LIN {X 0,Y 269.134,Z 589.137,A -85,B 0,C 180,E1 -17739.772,E2 -17739.772} C_VEL
LIN {X 0,Y 269.562,Z 582.717,A -85,B 0,C 180,E1 -17742.421,E2 -17742.421} C_VEL
LIN {X 0,Y 270.303,Z 575.756,A -85,B 0,C 180,E1 -17744.685,E2 -17744.685} C_VEL
LIN {X 0,Y 271.369,Z 568.724,A -85,B 0,C 180,E1 -17746.551,E2 -17746.551} C_VEL
LIN {X 0,Y 272.807,Z 560.299,A -85,B 0,C 180,E1 -17748.396,E2 -17748.396} C_VEL
LIN {X 0,Y 273.728,Z 553.275,A -85,B 0,C 180,E1 -17749.693,E2 -17749.693} C_VEL
LIN {X 0,Y 274.219,Z 542.305,A -85,B 0,C 180,E1 -17751.421,E2 -17751.421} C_VEL
LIN {X 0,Y 274.396,Z 531.867,A -85,B 0,C 180,E1 -17752.772,E2 -17752.772} C_VEL
LIN {X 0,Y 274.061,Z 519.052,A -85,B 0,C 180,E1 -17754.123,E2 -17754.123} C_VEL
LIN {X 0,Y 272.996,Z 505.88,A -85,B 0,C 180,E1 -17755.219,E2 -17755.219} C_VEL
LIN {X 0,Y 270.997,Z 492.141,A -85,B 0,C 180,E1 -17756.117,E2 -17756.117} C_VEL
LIN {X 0,Y 270.32,Z 487.569,A -85,B 0,C 180,E1 -17756.386,E2 -17756.386} C_VEL
LIN {X 0,Y 271.834,Z 476.288,A -85,B 0,C 180,E1 -17761.441,E2 -17761.441} C_VEL
LIN {X 0,Y 273.235,Z 467.638,A -85,B 0,C 180,E1 -17765.36,E2 -17765.36} C_VEL
LIN {X 0,Y 274.283,Z 461.982,A -85,B 0,C 180,E1 -17767.948,E2 -17767.948} C_VEL
LIN {X 0,Y 274.444,Z 460.134,A -85,B 0,C 180,E1 -17768.812,E2 -17768.812} C_VEL
LIN {X 0,Y 273.389,Z 453.927,A -85,B 0,C 180,E1 -17771.942,E2 -17771.942} C_VEL
LIN {X 0,Y 272.317,Z 448.311,A -85,B 0,C 180,E1 -17774.934,E2 -17774.934} C_VEL
LIN {X 0,Y 270.924,Z 441.471,A -85,B 0,C 180,E1 -17778.788,E2 -17778.788} C_VEL
LIN {X 0,Y 270.195,Z 437.829,A -85,B 0,C 180,E1 -17781.026,E2 -17781.026} C_VEL
LIN {X 0,Y 270.255,Z 437.821,A -85,B 0,C 180,E1 -17783.722,E2 -17783.722} C_VEL
LIN {X 0,Y 270.204,Z 437.829,A -85,B 0,C 180,E1 -17786.893,E2 -17786.893} C_VEL
LIN {X 0,Y 270.195,Z 437.83,A -85,B 0,C 180,E1 -17790.383,E2 -17790.383} C_VEL
LIN {X 0,Y 270.262,Z 437.819,A -85,B 0,C 180,E1 -17793.764,E2 -17793.764} C_VEL
LIN {X 0,Y 270.237,Z 437.822,A -85,B 0,C 180,E1 -17797.039,E2 -17797.039} C_VEL
LIN {X 0,Y 270.303,Z 437.818,A -85,B 0,C 180,E1 -17800.245,E2 -17800.245} C_VEL
LIN {X 0,Y 270.404,Z 437.802,A -85,B 0,C 180,E1 -17804.936,E2 -17804.936} C_VEL
LIN {X 0,Y 270.413,Z 437.801,A -85,B 0,C 180,E1 -17809.518,E2 -17809.518} C_VEL
LIN {X 0,Y 270.586,Z 437.779,A -85,B 0,C 180,E1 -17812.538,E2 -17812.538} C_VEL
LIN {X 0,Y 270.789,Z 437.753,A -85,B 0,C 180,E1 -17818.513,E2 -17818.513} C_VEL
LIN {X 0,Y 270.788,Z 437.752,A -85,B 0,C 180,E1 -17821.487,E2 -17821.487} C_VEL
LIN {X 0,Y 270.613,Z 437.771,A -85,B 0,C 180,E1 -17827.461,E2 -17827.461} C_VEL
LIN {X 0,Y 270.443,Z 437.795,A -85,B 0,C 180,E1 -17830.481,E2 -17830.481} C_VEL
LIN {X 0,Y 270.404,Z 437.798,A -85,B 0,C 180,E1 -17835.065,E2 -17835.065} C_VEL
LIN {X 0,Y 270.303,Z 437.806,A -85,B 0,C 180,E1 -17839.756,E2 -17839.756} C_VEL
LIN {X 0,Y 270.275,Z 437.81,A -85,B 0,C 180,E1 -17844.586,E2 -17844.586} C_VEL
LIN {X 0,Y 270.271,Z 437.821,A -85,B 0,C 180,E1 -17847.909,E2 -17847.909} C_VEL
LIN {X 0,Y 270.185,Z 437.823,A -85,B 0,C 180,E1 -17851.349,E2 -17851.349} C_VEL
LIN {X 0,Y 270.216,Z 437.817,A -85,B 0,C 180,E1 -17854.904,E2 -17854.904} C_VEL
LIN {X 0,Y 270.223,Z 437.822,A -85,B 0,C 180,E1 -17858.717,E2 -17858.717} C_VEL
LIN {X 0,Y 270.166,Z 437.829,A -85,B 0,C 180,E1 -17863.249,E2 -17863.249} C_VEL
LIN {X 0,Y 270.173,Z 437.829,A -85,B 0,C 180,E1 -17867.442,E2 -17867.442} C_VEL
LIN {X 0,Y 270.209,Z 437.823,A -85,B 0,C 180,E1 -17871.375,E2 -17871.375} C_VEL
LIN {X 0,Y 270.217,Z 437.819,A -85,B 0,C 180,E1 -17875.097,E2 -17875.097} C_VEL
LIN {X 0,Y 270.203,Z 437.825,A -85,B 0,C 180,E1 -17879.131,E2 -17879.131} C_VEL
LIN {X 0,Y 270.273,Z 437.816,A -85,B 0,C 180,E1 -17882.144,E2 -17882.144} C_VEL
LIN {X 0,Y 270.28,Z 437.813,A -85,B 0,C 180,E1 -17885.519,E2 -17885.519} C_VEL
LIN {X 0,Y 270.267,Z 437.861,A -85,B 0,C 180,E1 -17887.826,E2 -17887.826} C_VEL
LIN {X 0,Y 274.013,Z 447.701,A -85,B 0,C 180,E1 -17889.063,E2 -17889.063} C_VEL
LIN {X 0,Y 277.349,Z 457.508,A -85,B 0,C 180,E1 -17890.474,E2 -17890.474} C_VEL
LIN {X 0,Y 279.974,Z 467.572,A -85,B 0,C 180,E1 -17892.105,E2 -17892.105} C_VEL
LIN {X 0,Y 278.962,Z 475.715,A -85,B 0,C 180,E1 -17893.348,E2 -17893.348} C_VEL
LIN {X 0,Y 277.223,Z 486.274,A -85,B 0,C 180,E1 -17895.315,E2 -17895.315} C_VEL
LIN {X 0,Y 275.79,Z 494.07,A -85,B 0,C 180,E1 -17897.116,E2 -17897.116} C_VEL
LIN {X 0,Y 274.344,Z 501.7,A -85,B 0,C 180,E1 -17899.297,E2 -17899.297} C_VEL
LIN {X 0,Y 273.311,Z 506.88,A -85,B 0,C 180,E1 -17901.125,E2 -17901.125} C_VEL
LIN {X 0,Y 272.448,Z 511.909,A -85,B 0,C 180,E1 -17903.334,E2 -17903.334} C_VEL
LIN {X 0,Y 271.535,Z 515.856,A -85,B 0,C 180,E1 -17905.547,E2 -17905.547} C_VEL
LIN {X 0,Y 271.094,Z 517.898,A -85,B 0,C 180,E1 -17907.028,E2 -17907.028} C_VEL
LIN {X 0,Y 270.698,Z 520.727,A -85,B 0,C 180,E1 -17910,E2 -17910} C_VEL
LIN {X 0,Y 270.688,Z 521.555,A -85,B 0,C 180,E1 -17911.488,E2 -17911.488} C_VEL
LIN {X 0,Y 270.509,Z 522.06,A -85,B 0,C 180,E1 -17914.471,E2 -17914.471} C_VEL
LIN {X 0,Y 271.194,Z 521.003,A -85,B 0,C 180,E1 -17917.445,E2 -17917.445} C_VEL
LIN {X 0,Y 271.754,Z 519.845,A -85,B 0,C 180,E1 -17918.927,E2 -17918.927} C_VEL
LIN {X 0,Y 272.834,Z 516.501,A -85,B 0,C 180,E1 -17921.802,E2 -17921.802} C_VEL
LIN {X 0,Y 273.931,Z 512.606,A -85,B 0,C 180,E1 -17924.107,E2 -17924.107} C_VEL
LIN {X 0,Y 275.118,Z 507.732,A -85,B 0,C 180,E1 -17926.32,E2 -17926.32} C_VEL
LIN {X 0,Y 276.586,Z 501.563,A -85,B 0,C 180,E1 -17928.52,E2 -17928.52} C_VEL
LIN {X 0,Y 278.443,Z 493.783,A -85,B 0,C 180,E1 -17930.694,E2 -17930.694} C_VEL
LIN {X 0,Y 280.202,Z 485.823,A -85,B 0,C 180,E1 -17932.489,E2 -17932.489} C_VEL
LIN {X 0,Y 281.896,Z 476.106,A -85,B 0,C 180,E1 -17934.291,E2 -17934.291} C_VEL
LIN {X 0,Y 282.425,Z 472.703,A -85,B 0,C 180,E1 -17934.83,E2 -17934.83} C_VEL
LIN {X 0,Y 279.934,Z 463.035,A -85,B 0,C 180,E1 -17936.62,E2 -17936.62} C_VEL
LIN {X 0,Y 276.46,Z 452.721,A -85,B 0,C 180,E1 -17938.332,E2 -17938.332} C_VEL
LIN {X 0,Y 272.01,Z 442.14,A -85,B 0,C 180,E1 -17939.923,E2 -17939.923} C_VEL
LIN {X 0,Y 270.458,Z 438.953,A -85,B 0,C 180,E1 -17940.387,E2 -17940.387} C_VEL
LIN {X 0,Y 270.228,Z 437.825,A -85,B 0,C 180,E1 -17940.537,E2 -17940.537} C_VEL
LIN {X 0,Y 270.219,Z 437.824,A -85,B 0,C 180,E1 -17944.904,E2 -17944.904} C_VEL
LIN {X 0,Y 270.226,Z 437.824,A -85,B 0,C 180,E1 -17948.717,E2 -17948.717} C_VEL
LIN {X 0,Y 270.169,Z 437.83,A -85,B 0,C 180,E1 -17953.249,E2 -17953.249} C_VEL
LIN {X 0,Y 270.175,Z 437.827,A -85,B 0,C 180,E1 -17957.442,E2 -17957.442} C_VEL
LIN {X 0,Y 270.21,Z 437.823,A -85,B 0,C 180,E1 -17961.374,E2 -17961.374} C_VEL
LIN {X 0,Y 270.218,Z 437.822,A -85,B 0,C 180,E1 -17965.097,E2 -17965.097} C_VEL
LIN {X 0,Y 270.204,Z 437.825,A -85,B 0,C 180,E1 -17969.13,E2 -17969.13} C_VEL
LIN {X 0,Y 270.269,Z 437.818,A -85,B 0,C 180,E1 -17972.145,E2 -17972.145} C_VEL
LIN {X 0,Y 270.242,Z 437.821,A -85,B 0,C 180,E1 -17975.537,E2 -17975.537} C_VEL
LIN {X 0,Y 270.36,Z 437.805,A -85,B 0,C 180,E1 -17980.841,E2 -17980.841} C_VEL
LIN {X 0,Y 270.415,Z 437.929,A -85,B 0,C 180,E1 -17980.993,E2 -17980.993} C_VEL
LIN {X 0,Y 273.457,Z 451.257,A -85,B 0,C 180,E1 -17982.473,E2 -17982.473} C_VEL
LIN {X 0,Y 274.58,Z 456.844,A -85,B 0,C 180,E1 -17983.195,E2 -17983.195} C_VEL
LIN {X 0,Y 273.669,Z 469.268,A -85,B 0,C 180,E1 -17984.929,E2 -17984.929} C_VEL
LIN {X 0,Y 272.809,Z 479.061,A -85,B 0,C 180,E1 -17986.593,E2 -17986.593} C_VEL
LIN {X 0,Y 271.9,Z 490.128,A -85,B 0,C 180,E1 -17988.897,E2 -17988.897} C_VEL
LIN {X 0,Y 271.19,Z 498.55,A -85,B 0,C 180,E1 -17991.054,E2 -17991.054} C_VEL
LIN {X 0,Y 270.61,Z 506.844,A -85,B 0,C 180,E1 -17993.663,E2 -17993.663} C_VEL
LIN {X 0,Y 270.176,Z 513.358,A -85,B 0,C 180,E1 -17996.271,E2 -17996.271} C_VEL
LIN {X 0,Y 270.262,Z 517.749,A -85,B 0,C 180,E1 -17998.51,E2 -17998.51} C_VEL
LIN {X 0,Y 270.571,Z 520.097,A -85,B 0,C 180,E1 -18000,E2 -18000} C_VEL
LIN {X 0,Y 270.747,Z 522.029,A -85,B 0,C 180,E1 -18001.487,E2 -18001.487} C_VEL
LIN {X 0,Y 271.393,Z 524.678,A -85,B 0,C 180,E1 -18004.455,E2 -18004.455} C_VEL
LIN {X 0,Y 271.923,Z 525.431,A -85,B 0,C 180,E1 -18005.934,E2 -18005.934} C_VEL
LIN {X 0,Y 273.501,Z 525.662,A -85,B 0,C 180,E1 -18008.869,E2 -18008.869} C_VEL
LIN {X 0,Y 275.601,Z 524.401,A -85,B 0,C 180,E1 -18011.771,E2 -18011.771} C_VEL
LIN {X 0,Y 276.765,Z 523.168,A -85,B 0,C 180,E1 -18013.211,E2 -18013.211} C_VEL
LIN {X 0,Y 279.498,Z 519.777,A -85,B 0,C 180,E1 -18015.867,E2 -18015.867} C_VEL
LIN {X 0,Y 280.197,Z 518.177,A -85,B 0,C 180,E1 -18017.024,E2 -18017.024} C_VEL
LIN {X 0,Y 279.908,Z 515.583,A -85,B 0,C 180,E1 -18018.982,E2 -18018.982} C_VEL
LIN {X 0,Y 279.846,Z 512.387,A -85,B 0,C 180,E1 -18020.895,E2 -18020.895} C_VEL
LIN {X 0,Y 280.862,Z 509.845,A -85,B 0,C 180,E1 -18021.959,E2 -18021.959} C_VEL
LIN {X 0,Y 285.102,Z 501.844,A -85,B 0,C 180,E1 -18024.387,E2 -18024.387} C_VEL
LIN {X 0,Y 288.996,Z 493.552,A -85,B 0,C 180,E1 -18026.348,E2 -18026.348} C_VEL
LIN {X 0,Y 289.688,Z 491.994,A -85,B 0,C 180,E1 -18026.668,E2 -18026.668} C_VEL
LIN {X 0,Y 289.831,Z 489.623,A -85,B 0,C 180,E1 -18027.434,E2 -18027.434} C_VEL
LIN {X 0,Y 289.235,Z 483.398,A -85,B 0,C 180,E1 -18029.77,E2 -18029.77} C_VEL
LIN {X 0,Y 288.163,Z 478.273,A -85,B 0,C 180,E1 -18031.983,E2 -18031.983} C_VEL
LIN {X 0,Y 286.822,Z 473.819,A -85,B 0,C 180,E1 -18034.303,E2 -18034.303} C_VEL
LIN {X 0,Y 285.403,Z 471.506,A -85,B 0,C 180,E1 -18036.228,E2 -18036.228} C_VEL
LIN {X 0,Y 284.095,Z 470.015,A -85,B 0,C 180,E1 -18038.203,E2 -18038.203} C_VEL
LIN {X 0,Y 282.968,Z 469.651,A -85,B 0,C 180,E1 -18040.222,E2 -18040.222} C_VEL
LIN {X 0,Y 281.985,Z 470.615,A -85,B 0,C 180,E1 -18042.293,E2 -18042.293} C_VEL
LIN {X 0,Y 281.387,Z 472.597,A -85,B 0,C 180,E1 -18044.374,E2 -18044.374} C_VEL
LIN {X 0,Y 281.101,Z 475.772,A -85,B 0,C 180,E1 -18046.473,E2 -18046.473} C_VEL
LIN {X 0,Y 281.308,Z 479.869,A -85,B 0,C 180,E1 -18048.547,E2 -18048.547} C_VEL
LIN {X 0,Y 281.488,Z 484.367,A -85,B 0,C 180,E1 -18050.198,E2 -18050.198} C_VEL
LIN {X 0,Y 281.102,Z 490.544,A -85,B 0,C 180,E1 -18051.779,E2 -18051.779} C_VEL
LIN {X 0,Y 281.145,Z 493.947,A -85,B 0,C 180,E1 -18052.692,E2 -18052.692} C_VEL
LIN {X 0,Y 280.667,Z 508.223,A -85,B 0,C 180,E1 -18055.919,E2 -18055.919} C_VEL
LIN {X 0,Y 279.754,Z 521.489,A -85,B 0,C 180,E1 -18058.666,E2 -18058.666} C_VEL
LIN {X 0,Y 278.399,Z 532.665,A -85,B 0,C 180,E1 -18060.925,E2 -18060.925} C_VEL
LIN {X 0,Y 276.661,Z 541.8,A -85,B 0,C 180,E1 -18062.79,E2 -18062.79} C_VEL
LIN {X 0,Y 273.354,Z 553.407,A -85,B 0,C 180,E1 -18065.304,E2 -18065.304} C_VEL
LIN {X 0,Y 269.883,Z 564.585,A -85,B 0,C 180,E1 -18068.217,E2 -18068.217} C_VEL
LIN {X 0,Y 266.722,Z 572.712,A -85,B 0,C 180,E1 -18070.769,E2 -18070.769} C_VEL
LIN {X 0,Y 264.622,Z 578.556,A -85,B 0,C 180,E1 -18073.013,E2 -18073.013} C_VEL
LIN {X 0,Y 262.894,Z 584.824,A -85,B 0,C 180,E1 -18076.078,E2 -18076.078} C_VEL
LIN {X 0,Y 262.029,Z 594.375,A -85,B 0,C 180,E1 -18082.293,E2 -18082.293} C_VEL
LIN {X 0,Y 262.433,Z 597.47,A -85,B 0,C 180,E1 -18085.392,E2 -18085.392} C_VEL
LIN {X 0,Y 263.066,Z 598.826,A -85,B 0,C 180,E1 -18088.469,E2 -18088.469} C_VEL
LIN {X 0,Y 263.49,Z 598.901,A -85,B 0,C 180,E1 -18090,E2 -18090} C_VEL
LIN {X 0,Y 263.075,Z 598.446,A -85,B 0,C 180,E1 -18091.53,E2 -18091.53} C_VEL
LIN {X 0,Y 262.734,Z 597.546,A -85,B 0,C 180,E1 -18093.066,E2 -18093.066} C_VEL
LIN {X 0,Y 262.536,Z 596.227,A -85,B 0,C 180,E1 -18094.606,E2 -18094.606} C_VEL
LIN {X 0,Y 262.182,Z 592.821,A -85,B 0,C 180,E1 -18097.335,E2 -18097.335} C_VEL
LIN {X 0,Y 262.066,Z 588.033,A -85,B 0,C 180,E1 -18100.038,E2 -18100.038} C_VEL
LIN {X 0,Y 262.569,Z 581.59,A -85,B 0,C 180,E1 -18102.757,E2 -18102.757} C_VEL
LIN {X 0,Y 263.347,Z 574.603,A -85,B 0,C 180,E1 -18105.082,E2 -18105.082} C_VEL
LIN {X 0,Y 264.607,Z 567.41,A -85,B 0,C 180,E1 -18107.027,E2 -18107.027} C_VEL
LIN {X 0,Y 266.024,Z 559.1,A -85,B 0,C 180,E1 -18108.882,E2 -18108.882} C_VEL
LIN {X 0,Y 266.735,Z 553.115,A -85,B 0,C 180,E1 -18110.031,E2 -18110.031} C_VEL
LIN {X 0,Y 267.308,Z 542.427,A -85,B 0,C 180,E1 -18111.785,E2 -18111.785} C_VEL
LIN {X 0,Y 267.521,Z 530.306,A -85,B 0,C 180,E1 -18113.412,E2 -18113.412} C_VEL
LIN {X 0,Y 267.214,Z 517.51,A -85,B 0,C 180,E1 -18114.782,E2 -18114.782} C_VEL
LIN {X 0,Y 266.029,Z 503.862,A -85,B 0,C 180,E1 -18115.946,E2 -18115.946} C_VEL
LIN {X 0,Y 264.013,Z 490.435,A -85,B 0,C 180,E1 -18116.843,E2 -18116.843} C_VEL
LIN {X 0,Y 263.384,Z 486.54,A -85,B 0,C 180,E1 -18117.083,E2 -18117.083} C_VEL
LIN {X 0,Y 264.969,Z 475.794,A -85,B 0,C 180,E1 -18122.037,E2 -18122.037} C_VEL
LIN {X 0,Y 266.215,Z 468.377,A -85,B 0,C 180,E1 -18125.506,E2 -18125.506} C_VEL
LIN {X 0,Y 267.341,Z 462.21,A -85,B 0,C 180,E1 -18128.423,E2 -18128.423} C_VEL
LIN {X 0,Y 267.076,Z 458.563,A -85,B 0,C 180,E1 -18130.26,E2 -18130.26} C_VEL
LIN {X 0,Y 265.602,Z 450.824,A -85,B 0,C 180,E1 -18134.403,E2 -18134.403} C_VEL
LIN {X 0,Y 264.198,Z 444.015,A -85,B 0,C 180,E1 -18138.315,E2 -18138.315} C_VEL
LIN {X 0,Y 263.159,Z 438.707,A -85,B 0,C 180,E1 -18141.647,E2 -18141.647} C_VEL
LIN {X 0,Y 263.188,Z 438.702,A -85,B 0,C 180,E1 -18144.022,E2 -18144.022} C_VEL
LIN {X 0,Y 263.133,Z 438.71,A -85,B 0,C 180,E1 -18147.712,E2 -18147.712} C_VEL
LIN {X 0,Y 263.196,Z 438.702,A -85,B 0,C 180,E1 -18151.785,E2 -18151.785} C_VEL
LIN {X 0,Y 263.226,Z 438.695,A -85,B 0,C 180,E1 -18155.2,E2 -18155.2} C_VEL
LIN {X 0,Y 263.269,Z 438.693,A -85,B 0,C 180,E1 -18159.694,E2 -18159.694} C_VEL
LIN {X 0,Y 263.352,Z 438.682,A -85,B 0,C 180,E1 -18164.522,E2 -18164.522} C_VEL
LIN {X 0,Y 263.356,Z 438.68,A -85,B 0,C 180,E1 -18169.234,E2 -18169.234} C_VEL
LIN {X 0,Y 263.546,Z 438.658,A -85,B 0,C 180,E1 -18172.338,E2 -18172.338} C_VEL
LIN {X 0,Y 263.753,Z 438.63,A -85,B 0,C 180,E1 -18178.473,E2 -18178.473} C_VEL
LIN {X 0,Y 263.753,Z 438.629,A -85,B 0,C 180,E1 -18181.527,E2 -18181.527} C_VEL
LIN {X 0,Y 263.574,Z 438.649,A -85,B 0,C 180,E1 -18187.662,E2 -18187.662} C_VEL
LIN {X 0,Y 263.375,Z 438.674,A -85,B 0,C 180,E1 -18190.766,E2 -18190.766} C_VEL
LIN {X 0,Y 263.352,Z 438.678,A -85,B 0,C 180,E1 -18195.478,E2 -18195.478} C_VEL
LIN {X 0,Y 263.265,Z 438.677,A -85,B 0,C 180,E1 -18200.307,E2 -18200.307} C_VEL
LIN {X 0,Y 263.209,Z 438.69,A -85,B 0,C 180,E1 -18205.292,E2 -18205.292} C_VEL
LIN {X 0,Y 263.176,Z 438.7,A -85,B 0,C 180,E1 -18208.73,E2 -18208.73} C_VEL
LIN {X 0,Y 263.134,Z 438.691,A -85,B 0,C 180,E1 -18212.289,E2 -18212.289} C_VEL
LIN {X 0,Y 263.189,Z 438.698,A -85,B 0,C 180,E1 -18215.978,E2 -18215.978} C_VEL
LIN {X 0,Y 263.116,Z 438.708,A -85,B 0,C 180,E1 -18219.871,E2 -18219.871} C_VEL
LIN {X 0,Y 263.124,Z 438.705,A -85,B 0,C 180,E1 -18223.985,E2 -18223.985} C_VEL
LIN {X 0,Y 263.126,Z 438.703,A -85,B 0,C 180,E1 -18228.407,E2 -18228.407} C_VEL
LIN {X 0,Y 263.167,Z 438.7,A -85,B 0,C 180,E1 -18232.105,E2 -18232.105} C_VEL
LIN {X 0,Y 263.186,Z 438.701,A -85,B 0,C 180,E1 -18235.891,E2 -18235.891} C_VEL
LIN {X 0,Y 263.156,Z 438.705,A -85,B 0,C 180,E1 -18239.508,E2 -18239.508} C_VEL
LIN {X 0,Y 263.2,Z 438.699,A -85,B 0,C 180,E1 -18243.004,E2 -18243.004} C_VEL
LIN {X 0,Y 263.201,Z 438.7,A -85,B 0,C 180,E1 -18247.118,E2 -18247.118} C_VEL
LIN {X 0,Y 265.506,Z 444.774,A -85,B 0,C 180,E1 -18247.891,E2 -18247.891} C_VEL
LIN {X 0,Y 269.502,Z 455.525,A -85,B 0,C 180,E1 -18249.44,E2 -18249.44} C_VEL
LIN {X 0,Y 272.313,Z 465.51,A -85,B 0,C 180,E1 -18251.042,E2 -18251.042} C_VEL
LIN {X 0,Y 273.33,Z 470.093,A -85,B 0,C 180,E1 -18251.846,E2 -18251.846} C_VEL
LIN {X 0,Y 271.785,Z 480.105,A -85,B 0,C 180,E1 -18253.475,E2 -18253.475} C_VEL
LIN {X 0,Y 270.111,Z 489.175,A -85,B 0,C 180,E1 -18255.305,E2 -18255.305} C_VEL
LIN {X 0,Y 268.419,Z 497.955,A -85,B 0,C 180,E1 -18257.526,E2 -18257.526} C_VEL
LIN {X 0,Y 266.995,Z 505.021,A -85,B 0,C 180,E1 -18259.766,E2 -18259.766} C_VEL
LIN {X 0,Y 266.136,Z 509.77,A -85,B 0,C 180,E1 -18261.649,E2 -18261.649} C_VEL
LIN {X 0,Y 265.108,Z 514.417,A -85,B 0,C 180,E1 -18263.913,E2 -18263.913} C_VEL
LIN {X 0,Y 264.312,Z 517.986,A -85,B 0,C 180,E1 -18266.189,E2 -18266.189} C_VEL
LIN {X 0,Y 263.798,Z 520.564,A -85,B 0,C 180,E1 -18268.474,E2 -18268.474} C_VEL
LIN {X 0,Y 263.663,Z 522.584,A -85,B 0,C 180,E1 -18271.528,E2 -18271.528} C_VEL
LIN {X 0,Y 263.495,Z 523.068,A -85,B 0,C 180,E1 -18274.59,E2 -18274.59} C_VEL
LIN {X 0,Y 264.223,Z 521.986,A -85,B 0,C 180,E1 -18277.643,E2 -18277.643} C_VEL
LIN {X 0,Y 264.811,Z 520.814,A -85,B 0,C 180,E1 -18279.163,E2 -18279.163} C_VEL
LIN {X 0,Y 265.909,Z 517.522,A -85,B 0,C 180,E1 -18282.062,E2 -18282.062} C_VEL
LIN {X 0,Y 267.105,Z 513.537,A -85,B 0,C 180,E1 -18284.476,E2 -18284.476} C_VEL
LIN {X 0,Y 268.369,Z 508.639,A -85,B 0,C 180,E1 -18286.743,E2 -18286.743} C_VEL
LIN {X 0,Y 269.905,Z 502.435,A -85,B 0,C 180,E1 -18288.995,E2 -18288.995} C_VEL
LIN {X 0,Y 271.86,Z 494.623,A -85,B 0,C 180,E1 -18291.219,E2 -18291.219} C_VEL
LIN {X 0,Y 273.695,Z 486.63,A -85,B 0,C 180,E1 -18293.054,E2 -18293.054} C_VEL
LIN {X 0,Y 275.495,Z 476.869,A -85,B 0,C 180,E1 -18294.893,E2 -18294.893} C_VEL
LIN {X 0,Y 275.841,Z 474.601,A -85,B 0,C 180,E1 -18295.263,E2 -18295.263} C_VEL
LIN {X 0,Y 273.522,Z 465.506,A -85,B 0,C 180,E1 -18297.03,E2 -18297.03} C_VEL
LIN {X 0,Y 270.404,Z 455.984,A -85,B 0,C 180,E1 -18298.702,E2 -18298.702} C_VEL
LIN {X 0,Y 265.903,Z 445.066,A -85,B 0,C 180,E1 -18300.462,E2 -18300.462} C_VEL
LIN {X 0,Y 263.251,Z 439.311,A -85,B 0,C 180,E1 -18301.316,E2 -18301.316} C_VEL
LIN {X 0,Y 263.151,Z 438.706,A -85,B 0,C 180,E1 -18301.426,E2 -18301.426} C_VEL
LIN {X 0,Y 263.177,Z 438.704,A -85,B 0,C 180,E1 -18304.122,E2 -18304.122} C_VEL
LIN {X 0,Y 263.169,Z 438.704,A -85,B 0,C 180,E1 -18307.896,E2 -18307.896} C_VEL
LIN {X 0,Y 263.127,Z 438.71,A -85,B 0,C 180,E1 -18311.893,E2 -18311.893} C_VEL
LIN {X 0,Y 263.128,Z 438.708,A -85,B 0,C 180,E1 -18316.151,E2 -18316.151} C_VEL
LIN {X 0,Y 263.119,Z 438.707,A -85,B 0,C 180,E1 -18320.129,E2 -18320.129} C_VEL
LIN {X 0,Y 263.191,Z 438.698,A -85,B 0,C 180,E1 -18324.022,E2 -18324.022} C_VEL
LIN {X 0,Y 263.137,Z 438.705,A -85,B 0,C 180,E1 -18327.712,E2 -18327.712} C_VEL
LIN {X 0,Y 263.205,Z 438.697,A -85,B 0,C 180,E1 -18331.783,E2 -18331.783} C_VEL
LIN {X 0,Y 263.205,Z 438.697,A -85,B 0,C 180,E1 -18335.212,E2 -18335.212} C_VEL
LIN {X 0,Y 263.336,Z 438.796,A -85,B 0,C 180,E1 -18340.816,E2 -18340.816} C_VEL
LIN {X 0,Y 266.459,Z 452.411,A -85,B 0,C 180,E1 -18342.362,E2 -18342.362} C_VEL
LIN {X 0,Y 267.526,Z 457.017,A -85,B 0,C 180,E1 -18342.968,E2 -18342.968} C_VEL
LIN {X 0,Y 266.632,Z 469.291,A -85,B 0,C 180,E1 -18344.717,E2 -18344.717} C_VEL
LIN {X 0,Y 265.767,Z 479.227,A -85,B 0,C 180,E1 -18346.426,E2 -18346.426} C_VEL
LIN {X 0,Y 264.915,Z 489.291,A -85,B 0,C 180,E1 -18348.523,E2 -18348.523} C_VEL
LIN {X 0,Y 264.168,Z 498.393,A -85,B 0,C 180,E1 -18350.815,E2 -18350.815} C_VEL
LIN {X 0,Y 263.646,Z 505.836,A -85,B 0,C 180,E1 -18353.11,E2 -18353.11} C_VEL
LIN {X 0,Y 263.088,Z 511.944,A -85,B 0,C 180,E1 -18355.403,E2 -18355.403} C_VEL
LIN {X 0,Y 263.248,Z 516.853,A -85,B 0,C 180,E1 -18357.705,E2 -18357.705} C_VEL
LIN {X 0,Y 263.497,Z 520.724,A -85,B 0,C 180,E1 -18360,E2 -18360} C_VEL
LIN {X 0,Y 263.704,Z 522.797,A -85,B 0,C 180,E1 -18361.527,E2 -18361.527} C_VEL
LIN {X 0,Y 264.001,Z 524.453,A -85,B 0,C 180,E1 -18363.052,E2 -18363.052} C_VEL
LIN {X 0,Y 264.954,Z 526.541,A -85,B 0,C 180,E1 -18366.09,E2 -18366.09} C_VEL
LIN {X 0,Y 265.712,Z 527.018,A -85,B 0,C 180,E1 -18367.599,E2 -18367.599} C_VEL
LIN {X 0,Y 267.669,Z 526.727,A -85,B 0,C 180,E1 -18370.591,E2 -18370.591} C_VEL
LIN {X 0,Y 270.099,Z 524.975,A -85,B 0,C 180,E1 -18373.543,E2 -18373.543} C_VEL
LIN {X 0,Y 273.187,Z 521.58,A -85,B 0,C 180,E1 -18376.438,E2 -18376.438} C_VEL
LIN {X 0,Y 275.819,Z 517.946,A -85,B 0,C 180,E1 -18378.572,E2 -18378.572} C_VEL
LIN {X 0,Y 279.428,Z 512.331,A -85,B 0,C 180,E1 -18381.061,E2 -18381.061} C_VEL
LIN {X 0,Y 280.862,Z 509.845,A -85,B 0,C 180,E1 -18381.959,E2 -18381.959} C_VEL
LIN {X 0,Y 282.053,Z 507.124,A -85,B 0,C 180,E1 -18382.995,E2 -18382.995} C_VEL
LIN {X 0,Y 282.817,Z 502.831,A -85,B 0,C 180,E1 -18384.789,E2 -18384.789} C_VEL
LIN {X 0,Y 283.263,Z 499.161,A -85,B 0,C 180,E1 -18386.207,E2 -18386.207} C_VEL
LIN {X 0,Y 284.422,Z 494.839,A -85,B 0,C 180,E1 -18387.515,E2 -18387.515} C_VEL
LIN {X 0,Y 284.484,Z 489.457,A -85,B 0,C 180,E1 -18389.61,E2 -18389.61} C_VEL
LIN {X 0,Y 283.833,Z 484.037,A -85,B 0,C 180,E1 -18392.057,E2 -18392.057} C_VEL
LIN {X 0,Y 282.987,Z 480.214,A -85,B 0,C 180,E1 -18394.136,E2 -18394.136} C_VEL
LIN {X 0,Y 282.61,Z 479.156,A -85,B 0,C 180,E1 -18394.887,E2 -18394.887} C_VEL
LIN {X 0,Y 281.418,Z 477.118,A -85,B 0,C 180,E1 -18396.95,E2 -18396.95} C_VEL
LIN {X 0,Y 280.337,Z 476.081,A -85,B 0,C 180,E1 -18398.997,E2 -18398.997} C_VEL
LIN {X 0,Y 279.362,Z 476.303,A -85,B 0,C 180,E1 -18400.998,E2 -18400.998} C_VEL
LIN {X 0,Y 278.562,Z 477.629,A -85,B 0,C 180,E1 -18402.974,E2 -18402.974} C_VEL
LIN {X 0,Y 278.019,Z 480.162,A -85,B 0,C 180,E1 -18405.057,E2 -18405.057} C_VEL
LIN {X 0,Y 277.834,Z 485.249,A -85,B 0,C 180,E1 -18407.911,E2 -18407.911} C_VEL
LIN {X 0,Y 277.784,Z 488.964,A -85,B 0,C 180,E1 -18409.377,E2 -18409.377} C_VEL
LIN {X 0,Y 276.768,Z 499.239,A -85,B 0,C 180,E1 -18412.159,E2 -18412.159} C_VEL
LIN {X 0,Y 275.666,Z 511.972,A -85,B 0,C 180,E1 -18415.222,E2 -18415.222} C_VEL
LIN {X 0,Y 274.254,Z 524.486,A -85,B 0,C 180,E1 -18417.983,E2 -18417.983} C_VEL
LIN {X 0,Y 272.193,Z 536.663,A -85,B 0,C 180,E1 -18420.621,E2 -18420.621} C_VEL
LIN {X 0,Y 269.971,Z 545.247,A -85,B 0,C 180,E1 -18422.51,E2 -18422.51} C_VEL
LIN {X 0,Y 266.509,Z 555.838,A -85,B 0,C 180,E1 -18425.043,E2 -18425.043} C_VEL
LIN {X 0,Y 263.311,Z 564.995,A -85,B 0,C 180,E1 -18427.645,E2 -18427.645} C_VEL
LIN {X 0,Y 260.01,Z 572.783,A -85,B 0,C 180,E1 -18430.252,E2 -18430.252} C_VEL
LIN {X 0,Y 257.704,Z 578.545,A -85,B 0,C 180,E1 -18432.651,E2 -18432.651} C_VEL
LIN {X 0,Y 255.921,Z 584.29,A -85,B 0,C 180,E1 -18435.69,E2 -18435.69} C_VEL
LIN {X 0,Y 254.939,Z 593.386,A -85,B 0,C 180,E1 -18442.077,E2 -18442.077} C_VEL
LIN {X 0,Y 255.082,Z 595.134,A -85,B 0,C 180,E1 -18443.672,E2 -18443.672} C_VEL
LIN {X 0,Y 255.357,Z 596.471,A -85,B 0,C 180,E1 -18445.264,E2 -18445.264} C_VEL
LIN {X 0,Y 256.002,Z 597.811,A -85,B 0,C 180,E1 -18448.427,E2 -18448.427} C_VEL
LIN {X 0,Y 256.46,Z 597.885,A -85,B 0,C 180,E1 -18450,E2 -18450} C_VEL
LIN {X 0,Y 256.013,Z 597.416,A -85,B 0,C 180,E1 -18451.573,E2 -18451.573} C_VEL
LIN {X 0,Y 255.671,Z 596.501,A -85,B 0,C 180,E1 -18453.151,E2 -18453.151} C_VEL
LIN {X 0,Y 255.455,Z 595.17,A -85,B 0,C 180,E1 -18454.734,E2 -18454.734} C_VEL
LIN {X 0,Y 255.109,Z 592,A -85,B 0,C 180,E1 -18457.358,E2 -18457.358} C_VEL
LIN {X 0,Y 255.026,Z 586.93,A -85,B 0,C 180,E1 -18460.319,E2 -18460.319} C_VEL
LIN {X 0,Y 255.555,Z 580.458,A -85,B 0,C 180,E1 -18463.113,E2 -18463.113} C_VEL
LIN {X 0,Y 256.402,Z 573.448,A -85,B 0,C 180,E1 -18465.5,E2 -18465.5} C_VEL
LIN {X 0,Y 257.762,Z 566.395,A -85,B 0,C 180,E1 -18467.453,E2 -18467.453} C_VEL
LIN {X 0,Y 259.275,Z 557.901,A -85,B 0,C 180,E1 -18469.393,E2 -18469.393} C_VEL
LIN {X 0,Y 260.065,Z 548.512,A -85,B 0,C 180,E1 -18471.189,E2 -18471.189} C_VEL
LIN {X 0,Y 260.573,Z 538.04,A -85,B 0,C 180,E1 -18472.848,E2 -18472.848} C_VEL
LIN {X 0,Y 260.703,Z 527.129,A -85,B 0,C 180,E1 -18474.274,E2 -18474.274} C_VEL
LIN {X 0,Y 260.261,Z 514.76,A -85,B 0,C 180,E1 -18475.598,E2 -18475.598} C_VEL
LIN {X 0,Y 258.977,Z 501.526,A -85,B 0,C 180,E1 -18476.746,E2 -18476.746} C_VEL
LIN {X 0,Y 256.843,Z 488.091,A -85,B 0,C 180,E1 -18477.651,E2 -18477.651} C_VEL
LIN {X 0,Y 256.505,Z 485.536,A -85,B 0,C 180,E1 -18477.805,E2 -18477.805} C_VEL
LIN {X 0,Y 258.212,Z 474.685,A -85,B 0,C 180,E1 -18482.981,E2 -18482.981} C_VEL
LIN {X 0,Y 259.946,Z 465.381,A -85,B 0,C 180,E1 -18487.468,E2 -18487.468} C_VEL
LIN {X 0,Y 260.345,Z 461.555,A -85,B 0,C 180,E1 -18489.373,E2 -18489.373} C_VEL
LIN {X 0,Y 259.16,Z 455,A -85,B 0,C 180,E1 -18492.929,E2 -18492.929} C_VEL
LIN {X 0,Y 258.095,Z 449.565,A -85,B 0,C 180,E1 -18496.023,E2 -18496.023} C_VEL
LIN {X 0,Y 256.804,Z 442.953,A -85,B 0,C 180,E1 -18500.021,E2 -18500.021} C_VEL
LIN {X 0,Y 256.135,Z 439.58,A -85,B 0,C 180,E1 -18502.241,E2 -18502.241} C_VEL
LIN {X 0,Y 256.123,Z 439.582,A -85,B 0,C 180,E1 -18505.406,E2 -18505.406} C_VEL
LIN {X 0,Y 256.092,Z 439.589,A -85,B 0,C 180,E1 -18508.572,E2 -18508.572} C_VEL
LIN {X 0,Y 256.138,Z 439.579,A -85,B 0,C 180,E1 -18512.196,E2 -18512.196} C_VEL
LIN {X 0,Y 256.168,Z 439.576,A -85,B 0,C 180,E1 -18515.699,E2 -18515.699} C_VEL
LIN {X 0,Y 256.219,Z 439.57,A -85,B 0,C 180,E1 -18519.109,E2 -18519.109} C_VEL
LIN {X 0,Y 256.301,Z 439.563,A -85,B 0,C 180,E1 -18524.085,E2 -18524.085} C_VEL
LIN {X 0,Y 256.297,Z 439.559,A -85,B 0,C 180,E1 -18527.328,E2 -18527.328} C_VEL
LIN {X 0,Y 256.505,Z 439.535,A -85,B 0,C 180,E1 -18532.126,E2 -18532.126} C_VEL
LIN {X 0,Y 256.502,Z 439.532,A -85,B 0,C 180,E1 -18536.859,E2 -18536.859} C_VEL
LIN {X 0,Y 256.775,Z 439.502,A -85,B 0,C 180,E1 -18540,E2 -18540} C_VEL
LIN {X 0,Y 256.5,Z 439.532,A -85,B 0,C 180,E1 -18543.142,E2 -18543.142} C_VEL
LIN {X 0,Y 256.541,Z 439.526,A -85,B 0,C 180,E1 -18547.873,E2 -18547.873} C_VEL
LIN {X 0,Y 256.311,Z 439.554,A -85,B 0,C 180,E1 -18551.066,E2 -18551.066} C_VEL
LIN {X 0,Y 256.301,Z 439.559,A -85,B 0,C 180,E1 -18555.915,E2 -18555.915} C_VEL
LIN {X 0,Y 256.168,Z 439.558,A -85,B 0,C 180,E1 -18560.895,E2 -18560.895} C_VEL
LIN {X 0,Y 256.189,Z 439.564,A -85,B 0,C 180,E1 -18565.139,E2 -18565.139} C_VEL
LIN {X 0,Y 256.112,Z 439.582,A -85,B 0,C 180,E1 -18569.6,E2 -18569.6} C_VEL
LIN {X 0,Y 256.086,Z 439.566,A -85,B 0,C 180,E1 -18573.291,E2 -18573.291} C_VEL
LIN {X 0,Y 256.129,Z 439.578,A -85,B 0,C 180,E1 -18577.275,E2 -18577.275} C_VEL
LIN {X 0,Y 256.058,Z 439.585,A -85,B 0,C 180,E1 -18581.203,E2 -18581.203} C_VEL
LIN {X 0,Y 256.059,Z 439.585,A -85,B 0,C 180,E1 -18585.531,E2 -18585.531} C_VEL
LIN {X 0,Y 256.058,Z 439.583,A -85,B 0,C 180,E1 -18588.798,E2 -18588.798} C_VEL
LIN {X 0,Y 256.147,Z 439.573,A -85,B 0,C 180,E1 -18592.87,E2 -18592.87} C_VEL
LIN {X 0,Y 256.088,Z 439.582,A -85,B 0,C 180,E1 -18596.71,E2 -18596.71} C_VEL
LIN {X 0,Y 256.145,Z 439.57,A -85,B 0,C 180,E1 -18601.403,E2 -18601.403} C_VEL
LIN {X 0,Y 256.171,Z 439.57,A -85,B 0,C 180,E1 -18605.7,E2 -18605.7} C_VEL
LIN {X 0,Y 256.162,Z 439.576,A -85,B 0,C 180,E1 -18606.372,E2 -18606.372} C_VEL
LIN {X 0,Y 257.532,Z 443.418,A -85,B 0,C 180,E1 -18606.867,E2 -18606.867} C_VEL
LIN {X 0,Y 261.96,Z 454.746,A -85,B 0,C 180,E1 -18608.525,E2 -18608.525} C_VEL
LIN {X 0,Y 265.027,Z 464.794,A -85,B 0,C 180,E1 -18610.175,E2 -18610.175} C_VEL
LIN {X 0,Y 266.645,Z 471.439,A -85,B 0,C 180,E1 -18611.379,E2 -18611.379} C_VEL
LIN {X 0,Y 265.096,Z 481.351,A -85,B 0,C 180,E1 -18613.045,E2 -18613.045} C_VEL
LIN {X 0,Y 263.34,Z 490.373,A -85,B 0,C 180,E1 -18614.918,E2 -18614.918} C_VEL
LIN {X 0,Y 261.578,Z 499.121,A -85,B 0,C 180,E1 -18617.194,E2 -18617.194} C_VEL
LIN {X 0,Y 260.107,Z 506.158,A -85,B 0,C 180,E1 -18619.492,E2 -18619.492} C_VEL
LIN {X 0,Y 259.2,Z 510.884,A -85,B 0,C 180,E1 -18621.424,E2 -18621.424} C_VEL
LIN {X 0,Y 258.13,Z 515.51,A -85,B 0,C 180,E1 -18623.748,E2 -18623.748} C_VEL
LIN {X 0,Y 257.303,Z 519.059,A -85,B 0,C 180,E1 -18626.085,E2 -18626.085} C_VEL
LIN {X 0,Y 256.777,Z 521.618,A -85,B 0,C 180,E1 -18628.432,E2 -18628.432} C_VEL
LIN {X 0,Y 256.647,Z 522.816,A -85,B 0,C 180,E1 -18630,E2 -18630} C_VEL
LIN {X 0,Y 256.638,Z 523.611,A -85,B 0,C 180,E1 -18631.57,E2 -18631.57} C_VEL
LIN {X 0,Y 256.483,Z 524.076,A -85,B 0,C 180,E1 -18634.716,E2 -18634.716} C_VEL
LIN {X 0,Y 256.775,Z 523.723,A -85,B 0,C 180,E1 -18636.286,E2 -18636.286} C_VEL
LIN {X 0,Y 257.256,Z 522.968,A -85,B 0,C 180,E1 -18637.851,E2 -18637.851} C_VEL
LIN {X 0,Y 257.873,Z 521.784,A -85,B 0,C 180,E1 -18639.412,E2 -18639.412} C_VEL
LIN {X 0,Y 259.077,Z 518.284,A -85,B 0,C 180,E1 -18642.534,E2 -18642.534} C_VEL
LIN {X 0,Y 260.293,Z 514.468,A -85,B 0,C 180,E1 -18644.863,E2 -18644.863} C_VEL
LIN {X 0,Y 261.633,Z 509.545,A -85,B 0,C 180,E1 -18647.187,E2 -18647.187} C_VEL
LIN {X 0,Y 263.251,Z 503.306,A -85,B 0,C 180,E1 -18649.495,E2 -18649.495} C_VEL
LIN {X 0,Y 265.314,Z 495.463,A -85,B 0,C 180,E1 -18651.769,E2 -18651.769} C_VEL
LIN {X 0,Y 267.225,Z 487.436,A -85,B 0,C 180,E1 -18653.646,E2 -18653.646} C_VEL
LIN {X 0,Y 269.102,Z 477.736,A -85,B 0,C 180,E1 -18655.506,E2 -18655.506} C_VEL
LIN {X 0,Y 269.282,Z 476.638,A -85,B 0,C 180,E1 -18655.69,E2 -18655.69} C_VEL
LIN {X 0,Y 267.204,Z 468.206,A -85,B 0,C 180,E1 -18657.414,E2 -18657.414} C_VEL
LIN {X 0,Y 264.087,Z 458.413,A -85,B 0,C 180,E1 -18659.226,E2 -18659.226} C_VEL
LIN {X 0,Y 259.674,Z 447.697,A -85,B 0,C 180,E1 -18661.058,E2 -18661.058} C_VEL
LIN {X 0,Y 256.221,Z 440.269,A -85,B 0,C 180,E1 -18662.231,E2 -18662.231} C_VEL
LIN {X 0,Y 256.091,Z 439.587,A -85,B 0,C 180,E1 -18662.32,E2 -18662.32} C_VEL
LIN {X 0,Y 256.124,Z 439.58,A -85,B 0,C 180,E1 -18665.187,E2 -18665.187} C_VEL
LIN {X 0,Y 256.092,Z 439.584,A -85,B 0,C 180,E1 -18669.139,E2 -18669.139} C_VEL
LIN {X 0,Y 256.065,Z 439.587,A -85,B 0,C 180,E1 -18673.327,E2 -18673.327} C_VEL
LIN {X 0,Y 256.075,Z 439.584,A -85,B 0,C 180,E1 -18677.819,E2 -18677.819} C_VEL
LIN {X 0,Y 256.092,Z 439.581,A -85,B 0,C 180,E1 -18680.861,E2 -18680.861} C_VEL
LIN {X 0,Y 256.124,Z 439.578,A -85,B 0,C 180,E1 -18684.813,E2 -18684.813} C_VEL
LIN {X 0,Y 256.096,Z 439.582,A -85,B 0,C 180,E1 -18688.572,E2 -18688.572} C_VEL
LIN {X 0,Y 256.145,Z 439.577,A -85,B 0,C 180,E1 -18692.196,E2 -18692.196} C_VEL
LIN {X 0,Y 256.147,Z 439.576,A -85,B 0,C 180,E1 -18695.697,E2 -18695.697} C_VEL
LIN {X 0,Y 256.292,Z 439.557,A -85,B 0,C 180,E1 -18700.632,E2 -18700.632} C_VEL
LIN {X 0,Y 259.171,Z 452.437,A -85,B 0,C 180,E1 -18702.125,E2 -18702.125} C_VEL
LIN {X 0,Y 260.423,Z 458.466,A -85,B 0,C 180,E1 -18702.933,E2 -18702.933} C_VEL
LIN {X 0,Y 259.47,Z 471.671,A -85,B 0,C 180,E1 -18704.888,E2 -18704.888} C_VEL
LIN {X 0,Y 258.343,Z 483.292,A -85,B 0,C 180,E1 -18707.03,E2 -18707.03} C_VEL
LIN {X 0,Y 257.585,Z 492.908,A -85,B 0,C 180,E1 -18709.186,E2 -18709.186} C_VEL
LIN {X 0,Y 256.812,Z 502.148,A -85,B 0,C 180,E1 -18711.739,E2 -18711.739} C_VEL
LIN {X 0,Y 256.324,Z 509.137,A -85,B 0,C 180,E1 -18714.098,E2 -18714.098} C_VEL
LIN {X 0,Y 256.039,Z 513.961,A -85,B 0,C 180,E1 -18716.065,E2 -18716.065} C_VEL
LIN {X 0,Y 256.104,Z 518.749,A -85,B 0,C 180,E1 -18718.427,E2 -18718.427} C_VEL
LIN {X 0,Y 256.534,Z 522.493,A -85,B 0,C 180,E1 -18720.785,E2 -18720.785} C_VEL
LIN {X 0,Y 256.965,Z 525.287,A -85,B 0,C 180,E1 -18723.135,E2 -18723.135} C_VEL
LIN {X 0,Y 257.405,Z 526.681,A -85,B 0,C 180,E1 -18724.698,E2 -18724.698} C_VEL
LIN {X 0,Y 258.779,Z 528.224,A -85,B 0,C 180,E1 -18727.804,E2 -18727.804} C_VEL
LIN {X 0,Y 260.873,Z 528.241,A -85,B 0,C 180,E1 -18730.87,E2 -18730.87} C_VEL
LIN {X 0,Y 263.427,Z 526.731,A -85,B 0,C 180,E1 -18733.893,E2 -18733.893} C_VEL
LIN {X 0,Y 265.033,Z 525.392,A -85,B 0,C 180,E1 -18735.377,E2 -18735.377} C_VEL
LIN {X 0,Y 268.525,Z 521.526,A -85,B 0,C 180,E1 -18738.305,E2 -18738.305} C_VEL
LIN {X 0,Y 271.527,Z 517.52,A -85,B 0,C 180,E1 -18740.452,E2 -18740.452} C_VEL
LIN {X 0,Y 275.528,Z 511.518,A -85,B 0,C 180,E1 -18742.901,E2 -18742.901} C_VEL
LIN {X 0,Y 279.876,Z 503.94,A -85,B 0,C 180,E1 -18745.27,E2 -18745.27} C_VEL
LIN {X 0,Y 284.422,Z 494.839,A -85,B 0,C 180,E1 -18747.515,E2 -18747.515} C_VEL
LIN {X 0,Y 284.817,Z 492.849,A -85,B 0,C 180,E1 -18748.17,E2 -18748.17} C_VEL
LIN {X 0,Y 284.324,Z 491.195,A -85,B 0,C 180,E1 -18749.085,E2 -18749.085} C_VEL
LIN {X 0,Y 282.602,Z 489.94,A -85,B 0,C 180,E1 -18750.425,E2 -18750.425} C_VEL
LIN {X 0,Y 280.198,Z 488.952,A -85,B 0,C 180,E1 -18752.054,E2 -18752.054} C_VEL
LIN {X 0,Y 279.052,Z 487.641,A -85,B 0,C 180,E1 -18753.28,E2 -18753.28} C_VEL
LIN {X 0,Y 278.925,Z 486.963,A -85,B 0,C 180,E1 -18753.682,E2 -18753.682} C_VEL
LIN {X 0,Y 278.676,Z 485.464,A -85,B 0,C 180,E1 -18754.626,E2 -18754.626} C_VEL
LIN {X 0,Y 278.032,Z 483.98,A -85,B 0,C 180,E1 -18756.012,E2 -18756.012} C_VEL
LIN {X 0,Y 277.098,Z 482.561,A -85,B 0,C 180,E1 -18758.163,E2 -18758.163} C_VEL
LIN {X 0,Y 276.204,Z 482.38,A -85,B 0,C 180,E1 -18760.239,E2 -18760.239} C_VEL
LIN {X 0,Y 275.381,Z 483.449,A -85,B 0,C 180,E1 -18762.258,E2 -18762.258} C_VEL
LIN {X 0,Y 274.728,Z 485.538,A -85,B 0,C 180,E1 -18764.251,E2 -18764.251} C_VEL
LIN {X 0,Y 274.281,Z 488.619,A -85,B 0,C 180,E1 -18766.224,E2 -18766.224} C_VEL
LIN {X 0,Y 274.018,Z 492.591,A -85,B 0,C 180,E1 -18768.175,E2 -18768.175} C_VEL
LIN {X 0,Y 273.936,Z 493.896,A -85,B 0,C 180,E1 -18768.683,E2 -18768.683} C_VEL
LIN {X 0,Y 272.177,Z 504.648,A -85,B 0,C 180,E1 -18771.704,E2 -18771.704} C_VEL
LIN {X 0,Y 270.509,Z 516.84,A -85,B 0,C 180,E1 -18774.793,E2 -18774.793} C_VEL
LIN {X 0,Y 268.326,Z 529.396,A -85,B 0,C 180,E1 -18777.743,E2 -18777.743} C_VEL
LIN {X 0,Y 265.846,Z 540.443,A -85,B 0,C 180,E1 -18780.328,E2 -18780.328} C_VEL
LIN {X 0,Y 263.039,Z 548.988,A -85,B 0,C 180,E1 -18782.355,E2 -18782.355} C_VEL
LIN {X 0,Y 259.158,Z 559.364,A -85,B 0,C 180,E1 -18785.144,E2 -18785.144} C_VEL
LIN {X 0,Y 256.264,Z 566.584,A -85,B 0,C 180,E1 -18787.421,E2 -18787.421} C_VEL
LIN {X 0,Y 253.31,Z 572.805,A -85,B 0,C 180,E1 -18789.707,E2 -18789.707} C_VEL
LIN {X 0,Y 250.455,Z 579.421,A -85,B 0,C 180,E1 -18792.745,E2 -18792.745} C_VEL
LIN {X 0,Y 248.973,Z 583.713,A -85,B 0,C 180,E1 -18795.282,E2 -18795.282} C_VEL
LIN {X 0,Y 247.818,Z 590.232,A -85,B 0,C 180,E1 -18800.203,E2 -18800.203} C_VEL
LIN {X 0,Y 247.949,Z 593.442,A -85,B 0,C 180,E1 -18802.775,E2 -18802.775} C_VEL
LIN {X 0,Y 248.284,Z 595.47,A -85,B 0,C 180,E1 -18805.128,E2 -18805.128} C_VEL
LIN {X 0,Y 248.937,Z 596.797,A -85,B 0,C 180,E1 -18808.382,E2 -18808.382} C_VEL
LIN {X 0,Y 249.429,Z 596.868,A -85,B 0,C 180,E1 -18810,E2 -18810} C_VEL
LIN {X 0,Y 248.951,Z 596.385,A -85,B 0,C 180,E1 -18811.617,E2 -18811.617} C_VEL
LIN {X 0,Y 248.606,Z 595.455,A -85,B 0,C 180,E1 -18813.241,E2 -18813.241} C_VEL
LIN {X 0,Y 248.377,Z 594.112,A -85,B 0,C 180,E1 -18814.869,E2 -18814.869} C_VEL
LIN {X 0,Y 248.059,Z 591.125,A -85,B 0,C 180,E1 -18817.424,E2 -18817.424} C_VEL
LIN {X 0,Y 247.934,Z 587.349,A -85,B 0,C 180,E1 -18819.792,E2 -18819.792} C_VEL
LIN {X 0,Y 248.251,Z 582.312,A -85,B 0,C 180,E1 -18822.258,E2 -18822.258} C_VEL
LIN {X 0,Y 248.966,Z 575.996,A -85,B 0,C 180,E1 -18824.718,E2 -18824.718} C_VEL
LIN {X 0,Y 250.083,Z 568.832,A -85,B 0,C 180,E1 -18826.971,E2 -18826.971} C_VEL
LIN {X 0,Y 251.53,Z 561.991,A -85,B 0,C 180,E1 -18828.743,E2 -18828.743} C_VEL
LIN {X 0,Y 252.713,Z 554.738,A -85,B 0,C 180,E1 -18830.342,E2 -18830.342} C_VEL
LIN {X 0,Y 253.464,Z 543.598,A -85,B 0,C 180,E1 -18832.411,E2 -18832.411} C_VEL
LIN {X 0,Y 253.868,Z 533.183,A -85,B 0,C 180,E1 -18833.998,E2 -18833.998} C_VEL
LIN {X 0,Y 253.827,Z 520.94,A -85,B 0,C 180,E1 -18835.524,E2 -18835.524} C_VEL
LIN {X 0,Y 253.013,Z 508.003,A -85,B 0,C 180,E1 -18836.832,E2 -18836.832} C_VEL
LIN {X 0,Y 251.246,Z 494.001,A -85,B 0,C 180,E1 -18837.966,E2 -18837.966} C_VEL
LIN {X 0,Y 249.627,Z 484.426,A -85,B 0,C 180,E1 -18838.595,E2 -18838.595} C_VEL
LIN {X 0,Y 251.243,Z 474.773,A -85,B 0,C 180,E1 -18843.367,E2 -18843.367} C_VEL
LIN {X 0,Y 252.947,Z 466.109,A -85,B 0,C 180,E1 -18847.68,E2 -18847.68} C_VEL
LIN {X 0,Y 253.306,Z 462.311,A -85,B 0,C 180,E1 -18849.653,E2 -18849.653} C_VEL
LIN {X 0,Y 252.015,Z 455.4,A -85,B 0,C 180,E1 -18853.525,E2 -18853.525} C_VEL
LIN {X 0,Y 250.656,Z 448.393,A -85,B 0,C 180,E1 -18857.707,E2 -18857.707} C_VEL
LIN {X 0,Y 249.289,Z 441.521,A -85,B 0,C 180,E1 -18862.127,E2 -18862.127} C_VEL
LIN {X 0,Y 249.119,Z 440.455,A -85,B 0,C 180,E1 -18862.888,E2 -18862.888} C_VEL
LIN {X 0,Y 249.036,Z 440.466,A -85,B 0,C 180,E1 -18867.575,E2 -18867.575} C_VEL
LIN {X 0,Y 249.086,Z 440.458,A -85,B 0,C 180,E1 -18871.337,E2 -18871.337} C_VEL
LIN {X 0,Y 249.152,Z 440.449,A -85,B 0,C 180,E1 -18874.969,E2 -18874.969} C_VEL
LIN {X 0,Y 249.127,Z 440.455,A -85,B 0,C 180,E1 -18878.582,E2 -18878.582} C_VEL
LIN {X 0,Y 249.242,Z 440.44,A -85,B 0,C 180,E1 -18883.622,E2 -18883.622} C_VEL
LIN {X 0,Y 249.246,Z 440.439,A -85,B 0,C 180,E1 -18888.616,E2 -18888.616} C_VEL
LIN {X 0,Y 249.447,Z 440.415,A -85,B 0,C 180,E1 -18891.902,E2 -18891.902} C_VEL
LIN {X 0,Y 249.299,Z 440.429,A -85,B 0,C 180,E1 -18895.149,E2 -18895.149} C_VEL
LIN {X 0,Y 249.678,Z 440.384,A -85,B 0,C 180,E1 -18898.387,E2 -18898.387} C_VEL
LIN {X 0,Y 249.677,Z 440.382,A -85,B 0,C 180,E1 -18901.613,E2 -18901.613} C_VEL
LIN {X 0,Y 249.452,Z 440.405,A -85,B 0,C 180,E1 -18906.772,E2 -18906.772} C_VEL
LIN {X 0,Y 249.425,Z 440.415,A -85,B 0,C 180,E1 -18909.734,E2 -18909.734} C_VEL
LIN {X 0,Y 249.207,Z 440.439,A -85,B 0,C 180,E1 -18914.704,E2 -18914.704} C_VEL
LIN {X 0,Y 249.141,Z 440.446,A -85,B 0,C 180,E1 -18918.078,E2 -18918.078} C_VEL
LIN {X 0,Y 249.088,Z 440.434,A -85,B 0,C 180,E1 -18921.518,E2 -18921.518} C_VEL
LIN {X 0,Y 249.132,Z 440.444,A -85,B 0,C 180,E1 -18925.483,E2 -18925.483} C_VEL
LIN {X 0,Y 249.081,Z 440.456,A -85,B 0,C 180,E1 -18928.992,E2 -18928.992} C_VEL
LIN {X 0,Y 249.037,Z 440.444,A -85,B 0,C 180,E1 -18932.425,E2 -18932.425} C_VEL
LIN {X 0,Y 249.07,Z 440.458,A -85,B 0,C 180,E1 -18936.339,E2 -18936.339} C_VEL
LIN {X 0,Y 249.027,Z 440.461,A -85,B 0,C 180,E1 -18940.475,E2 -18940.475} C_VEL
LIN {X 0,Y 249.004,Z 440.461,A -85,B 0,C 180,E1 -18944.88,E2 -18944.88} C_VEL
LIN {X 0,Y 249.018,Z 440.463,A -85,B 0,C 180,E1 -18947.363,E2 -18947.363} C_VEL
LIN {X 0,Y 249.04,Z 440.458,A -85,B 0,C 180,E1 -18951.622,E2 -18951.622} C_VEL
LIN {X 0,Y 249.064,Z 440.457,A -85,B 0,C 180,E1 -18955.643,E2 -18955.643} C_VEL
LIN {X 0,Y 249.056,Z 440.461,A -85,B 0,C 180,E1 -18959.474,E2 -18959.474} C_VEL
LIN {X 0,Y 249.079,Z 440.458,A -85,B 0,C 180,E1 -18963.163,E2 -18963.163} C_VEL
LIN {X 0,Y 249.135,Z 440.446,A -85,B 0,C 180,E1 -18965.591,E2 -18965.591} C_VEL
LIN {X 0,Y 251.364,Z 446.357,A -85,B 0,C 180,E1 -18966.396,E2 -18966.396} C_VEL
LIN {X 0,Y 255.257,Z 456.49,A -85,B 0,C 180,E1 -18967.968,E2 -18967.968} C_VEL
LIN {X 0,Y 258.127,Z 465.428,A -85,B 0,C 180,E1 -18969.504,E2 -18969.504} C_VEL
LIN {X 0,Y 259.926,Z 472.799,A -85,B 0,C 180,E1 -18970.885,E2 -18970.885} C_VEL
LIN {X 0,Y 258.415,Z 482.591,A -85,B 0,C 180,E1 -18972.593,E2 -18972.593} C_VEL
LIN {X 0,Y 256.58,Z 491.571,A -85,B 0,C 180,E1 -18974.511,E2 -18974.511} C_VEL
LIN {X 0,Y 254.763,Z 500.285,A -85,B 0,C 180,E1 -18976.845,E2 -18976.845} C_VEL
LIN {X 0,Y 253.221,Z 507.295,A -85,B 0,C 180,E1 -18979.203,E2 -18979.203} C_VEL
LIN {X 0,Y 252.268,Z 511.999,A -85,B 0,C 180,E1 -18981.186,E2 -18981.186} C_VEL
LIN {X 0,Y 251.154,Z 516.604,A -85,B 0,C 180,E1 -18983.574,E2 -18983.574} C_VEL
LIN {X 0,Y 250.541,Z 519.09,A -85,B 0,C 180,E1 -18985.173,E2 -18985.173} C_VEL
LIN {X 0,Y 250.055,Z 521.087,A -85,B 0,C 180,E1 -18986.778,E2 -18986.778} C_VEL
LIN {X 0,Y 249.622,Z 523.86,A -85,B 0,C 180,E1 -18990,E2 -18990} C_VEL
LIN {X 0,Y 249.613,Z 524.636,A -85,B 0,C 180,E1 -18991.614,E2 -18991.614} C_VEL
LIN {X 0,Y 249.473,Z 525.084,A -85,B 0,C 180,E1 -18994.848,E2 -18994.848} C_VEL
LIN {X 0,Y 249.785,Z 524.721,A -85,B 0,C 180,E1 -18996.462,E2 -18996.462} C_VEL
LIN {X 0,Y 250.293,Z 523.948,A -85,B 0,C 180,E1 -18998.071,E2 -18998.071} C_VEL
LIN {X 0,Y 250.94,Z 522.754,A -85,B 0,C 180,E1 -18999.674,E2 -18999.674} C_VEL
LIN {X 0,Y 252.08,Z 519.564,A -85,B 0,C 180,E1 -19002.628,E2 -19002.628} C_VEL
LIN {X 0,Y 253.495,Z 515.398,A -85,B 0,C 180,E1 -19005.271,E2 -19005.271} C_VEL
LIN {X 0,Y 254.912,Z 510.449,A -85,B 0,C 180,E1 -19007.655,E2 -19007.655} C_VEL
LIN {X 0,Y 256.62,Z 504.177,A -85,B 0,C 180,E1 -19010.02,E2 -19010.02} C_VEL
LIN {X 0,Y 258.798,Z 496.302,A -85,B 0,C 180,E1 -19012.346,E2 -19012.346} C_VEL
LIN {X 0,Y 260.771,Z 488.243,A -85,B 0,C 180,E1 -19014.268,E2 -19014.268} C_VEL
LIN {X 0,Y 262.661,Z 478.91,A -85,B 0,C 180,E1 -19016.096,E2 -19016.096} C_VEL
LIN {X 0,Y 261.068,Z 471.606,A -85,B 0,C 180,E1 -19017.656,E2 -19017.656} C_VEL
LIN {X 0,Y 257.934,Z 461.354,A -85,B 0,C 180,E1 -19019.684,E2 -19019.684} C_VEL
LIN {X 0,Y 253.708,Z 450.876,A -85,B 0,C 180,E1 -19021.59,E2 -19021.59} C_VEL
LIN {X 0,Y 249.147,Z 441.022,A -85,B 0,C 180,E1 -19023.232,E2 -19023.232} C_VEL
LIN {X 0,Y 249.051,Z 440.463,A -85,B 0,C 180,E1 -19023.343,E2 -19023.343} C_VEL
LIN {X 0,Y 249.073,Z 440.46,A -85,B 0,C 180,E1 -19026.339,E2 -19026.339} C_VEL
LIN {X 0,Y 249.029,Z 440.465,A -85,B 0,C 180,E1 -19030.474,E2 -19030.474} C_VEL
LIN {X 0,Y 249.006,Z 440.466,A -85,B 0,C 180,E1 -19034.879,E2 -19034.879} C_VEL
LIN {X 0,Y 249.02,Z 440.462,A -85,B 0,C 180,E1 -19037.363,E2 -19037.363} C_VEL
LIN {X 0,Y 249.042,Z 440.46,A -85,B 0,C 180,E1 -19041.622,E2 -19041.622} C_VEL
LIN {X 0,Y 249.065,Z 440.459,A -85,B 0,C 180,E1 -19045.642,E2 -19045.642} C_VEL
LIN {X 0,Y 249.056,Z 440.46,A -85,B 0,C 180,E1 -19049.473,E2 -19049.473} C_VEL
LIN {X 0,Y 249.074,Z 440.457,A -85,B 0,C 180,E1 -19053.162,E2 -19053.162} C_VEL
LIN {X 0,Y 249.065,Z 440.458,A -85,B 0,C 180,E1 -19056.731,E2 -19056.731} C_VEL
LIN {X 0,Y 249.258,Z 440.517,A -85,B 0,C 180,E1 -19060.464,E2 -19060.464} C_VEL
LIN {X 0,Y 252.176,Z 453.645,A -85,B 0,C 180,E1 -19062.031,E2 -19062.031} C_VEL
LIN {X 0,Y 253.264,Z 458.081,A -85,B 0,C 180,E1 -19062.644,E2 -19062.644} C_VEL
LIN {X 0,Y 252.698,Z 467.89,A -85,B 0,C 180,E1 -19064.059,E2 -19064.059} C_VEL
LIN {X 0,Y 251.82,Z 478.352,A -85,B 0,C 180,E1 -19065.865,E2 -19065.865} C_VEL
LIN {X 0,Y 250.795,Z 489.814,A -85,B 0,C 180,E1 -19068.278,E2 -19068.278} C_VEL
LIN {X 0,Y 250.01,Z 499.135,A -85,B 0,C 180,E1 -19070.698,E2 -19070.698} C_VEL
LIN {X 0,Y 249.431,Z 506.868,A -85,B 0,C 180,E1 -19073.122,E2 -19073.122} C_VEL
LIN {X 0,Y 248.963,Z 514.164,A -85,B 0,C 180,E1 -19075.953,E2 -19075.953} C_VEL
LIN {X 0,Y 249.024,Z 519.145,A -85,B 0,C 180,E1 -19078.383,E2 -19078.383} C_VEL
LIN {X 0,Y 249.47,Z 523.07,A -85,B 0,C 180,E1 -19080.807,E2 -19080.807} C_VEL
LIN {X 0,Y 249.932,Z 526.074,A -85,B 0,C 180,E1 -19083.224,E2 -19083.224} C_VEL
LIN {X 0,Y 251.019,Z 528.724,A -85,B 0,C 180,E1 -19086.43,E2 -19086.43} C_VEL
LIN {X 0,Y 252.897,Z 529.743,A -85,B 0,C 180,E1 -19089.598,E2 -19089.598} C_VEL
LIN {X 0,Y 255.392,Z 529.284,A -85,B 0,C 180,E1 -19092.718,E2 -19092.718} C_VEL
LIN {X 0,Y 258.445,Z 527.295,A -85,B 0,C 180,E1 -19095.779,E2 -19095.779} C_VEL
LIN {X 0,Y 260.21,Z 525.751,A -85,B 0,C 180,E1 -19097.283,E2 -19097.283} C_VEL
LIN {X 0,Y 263.154,Z 522.629,A -85,B 0,C 180,E1 -19099.502,E2 -19099.502} C_VEL
LIN {X 0,Y 266.466,Z 518.608,A -85,B 0,C 180,E1 -19101.669,E2 -19101.669} C_VEL
LIN {X 0,Y 270.13,Z 513.522,A -85,B 0,C 180,E1 -19103.782,E2 -19103.782} C_VEL
LIN {X 0,Y 274.837,Z 506.038,A -85,B 0,C 180,E1 -19106.216,E2 -19106.216} C_VEL
LIN {X 0,Y 279.223,Z 498.145,A -85,B 0,C 180,E1 -19108.242,E2 -19108.242} C_VEL
LIN {X 0,Y 279.437,Z 492.541,A -85,B 0,C 180,E1 -19110.711,E2 -19110.711} C_VEL
LIN {X 0,Y 279.143,Z 488.622,A -85,B 0,C 180,E1 -19112.701,E2 -19112.701} C_VEL
LIN {X 0,Y 278.925,Z 486.963,A -85,B 0,C 180,E1 -19113.682,E2 -19113.682} C_VEL
LIN {X 0,Y 278.611,Z 485.9,A -85,B 0,C 180,E1 -19114.454,E2 -19114.454} C_VEL
LIN {X 0,Y 277.509,Z 485.42,A -85,B 0,C 180,E1 -19115.647,E2 -19115.647} C_VEL
LIN {X 0,Y 276.014,Z 485.873,A -85,B 0,C 180,E1 -19116.84,E2 -19116.84} C_VEL
LIN {X 0,Y 273.088,Z 487.909,A -85,B 0,C 180,E1 -19119.311,E2 -19119.311} C_VEL
LIN {X 0,Y 272.506,Z 488.429,A -85,B 0,C 180,E1 -19120.159,E2 -19120.159} C_VEL
LIN {X 0,Y 271.661,Z 489.665,A -85,B 0,C 180,E1 -19122.271,E2 -19122.271} C_VEL
LIN {X 0,Y 271.255,Z 490.86,A -85,B 0,C 180,E1 -19123.492,E2 -19123.492} C_VEL
LIN {X 0,Y 270.451,Z 494.714,A -85,B 0,C 180,E1 -19126.056,E2 -19126.056} C_VEL
LIN {X 0,Y 270.129,Z 497.434,A -85,B 0,C 180,E1 -19127.433,E2 -19127.433} C_VEL
LIN {X 0,Y 269.794,Z 499.162,A -85,B 0,C 180,E1 -19128.102,E2 -19128.102} C_VEL
LIN {X 0,Y 267.675,Z 508.792,A -85,B 0,C 180,E1 -19130.939,E2 -19130.939} C_VEL
LIN {X 0,Y 265.4,Z 520.145,A -85,B 0,C 180,E1 -19134.011,E2 -19134.011} C_VEL
LIN {X 0,Y 263.026,Z 530.75,A -85,B 0,C 180,E1 -19136.678,E2 -19136.678} C_VEL
LIN {X 0,Y 259.968,Z 542.138,A -85,B 0,C 180,E1 -19139.543,E2 -19139.543} C_VEL
LIN {X 0,Y 256.064,Z 552.363,A -85,B 0,C 180,E1 -19142.187,E2 -19142.187} C_VEL
LIN {X 0,Y 251.244,Z 563.675,A -85,B 0,C 180,E1 -19145.631,E2 -19145.631} C_VEL
LIN {X 0,Y 247.591,Z 570.985,A -85,B 0,C 180,E1 -19148.345,E2 -19148.345} C_VEL
LIN {X 0,Y 244.236,Z 577.818,A -85,B 0,C 180,E1 -19151.546,E2 -19151.546} C_VEL
LIN {X 0,Y 242.046,Z 583.142,A -85,B 0,C 180,E1 -19154.851,E2 -19154.851} C_VEL
LIN {X 0,Y 240.828,Z 587.992,A -85,B 0,C 180,E1 -19159.065,E2 -19159.065} C_VEL
LIN {X 0,Y 240.799,Z 591.413,A -85,B 0,C 180,E1 -19161.608,E2 -19161.608} C_VEL
LIN {X 0,Y 240.946,Z 593.153,A -85,B 0,C 180,E1 -19163.299,E2 -19163.299} C_VEL
LIN {X 0,Y 241.213,Z 594.469,A -85,B 0,C 180,E1 -19164.985,E2 -19164.985} C_VEL
LIN {X 0,Y 241.872,Z 595.783,A -85,B 0,C 180,E1 -19168.335,E2 -19168.335} C_VEL
LIN {X 0,Y 242.394,Z 595.851,A -85,B 0,C 180,E1 -19170,E2 -19170} C_VEL
LIN {X 0,Y 241.888,Z 595.352,A -85,B 0,C 180,E1 -19171.665,E2 -19171.665} C_VEL
LIN {X 0,Y 241.541,Z 594.409,A -85,B 0,C 180,E1 -19173.336,E2 -19173.336} C_VEL
LIN {X 0,Y 241.302,Z 593.055,A -85,B 0,C 180,E1 -19175.012,E2 -19175.012} C_VEL
LIN {X 0,Y 240.986,Z 590.305,A -85,B 0,C 180,E1 -19177.45,E2 -19177.45} C_VEL
LIN {X 0,Y 240.871,Z 586.248,A -85,B 0,C 180,E1 -19180.082,E2 -19180.082} C_VEL
LIN {X 0,Y 241.25,Z 581.192,A -85,B 0,C 180,E1 -19182.62,E2 -19182.62} C_VEL
LIN {X 0,Y 242.004,Z 574.85,A -85,B 0,C 180,E1 -19185.151,E2 -19185.151} C_VEL
LIN {X 0,Y 243.42,Z 567.311,A -85,B 0,C 180,E1 -19187.568,E2 -19187.568} C_VEL
LIN {X 0,Y 245.083,Z 559.125,A -85,B 0,C 180,E1 -19189.69,E2 -19189.69} C_VEL
LIN {X 0,Y 246.003,Z 551.454,A -85,B 0,C 180,E1 -19191.361,E2 -19191.361} C_VEL
LIN {X 0,Y 246.744,Z 541.053,A -85,B 0,C 180,E1 -19193.278,E2 -19193.278} C_VEL
LIN {X 0,Y 247.116,Z 528.815,A -85,B 0,C 180,E1 -19195.111,E2 -19195.111} C_VEL
LIN {X 0,Y 246.891,Z 516.633,A -85,B 0,C 180,E1 -19196.601,E2 -19196.601} C_VEL
LIN {X 0,Y 246.023,Z 505.101,A -85,B 0,C 180,E1 -19197.762,E2 -19197.762} C_VEL
LIN {X 0,Y 244.289,Z 492.356,A -85,B 0,C 180,E1 -19198.813,E2 -19198.813} C_VEL
LIN {X 0,Y 242.77,Z 483.335,A -85,B 0,C 180,E1 -19199.42,E2 -19199.42} C_VEL
LIN {X 0,Y 244.428,Z 474.101,A -85,B 0,C 180,E1 -19204.157,E2 -19204.157} C_VEL
LIN {X 0,Y 245.962,Z 466.833,A -85,B 0,C 180,E1 -19207.903,E2 -19207.903} C_VEL
LIN {X 0,Y 246.296,Z 463.609,A -85,B 0,C 180,E1 -19209.607,E2 -19209.607} C_VEL
LIN {X 0,Y 245.088,Z 456.897,A -85,B 0,C 180,E1 -19213.488,E2 -19213.488} C_VEL
LIN {X 0,Y 243.852,Z 450.571,A -85,B 0,C 180,E1 -19217.368,E2 -19217.368} C_VEL
LIN {X 0,Y 242.613,Z 444.331,A -85,B 0,C 180,E1 -19221.456,E2 -19221.456} C_VEL
LIN {X 0,Y 242.035,Z 441.336,A -85,B 0,C 180,E1 -19223.599,E2 -19223.599} C_VEL
LIN {X 0,Y 241.995,Z 441.343,A -85,B 0,C 180,E1 -19227.374,E2 -19227.374} C_VEL
LIN {X 0,Y 242.014,Z 441.34,A -85,B 0,C 180,E1 -19230.597,E2 -19230.597} C_VEL
LIN {X 0,Y 242.068,Z 441.334,A -85,B 0,C 180,E1 -19234.183,E2 -19234.183} C_VEL
LIN {X 0,Y 242.065,Z 441.335,A -85,B 0,C 180,E1 -19238.29,E2 -19238.29} C_VEL
LIN {X 0,Y 242.163,Z 441.321,A -85,B 0,C 180,E1 -19243.278,E2 -19243.278} C_VEL
LIN {X 0,Y 242.182,Z 441.321,A -85,B 0,C 180,E1 -19248.28,E2 -19248.28} C_VEL
LIN {X 0,Y 242.394,Z 441.293,A -85,B 0,C 180,E1 -19251.665,E2 -19251.665} C_VEL
LIN {X 0,Y 242.259,Z 441.306,A -85,B 0,C 180,E1 -19255.007,E2 -19255.007} C_VEL
LIN {X 0,Y 242.638,Z 441.261,A -85,B 0,C 180,E1 -19258.34,E2 -19258.34} C_VEL
LIN {X 0,Y 242.638,Z 441.26,A -85,B 0,C 180,E1 -19261.66,E2 -19261.66} C_VEL
LIN {X 0,Y 242.43,Z 441.28,A -85,B 0,C 180,E1 -19266.751,E2 -19266.751} C_VEL
LIN {X 0,Y 242.346,Z 441.298,A -85,B 0,C 180,E1 -19270.021,E2 -19270.021} C_VEL
LIN {X 0,Y 242.168,Z 441.316,A -85,B 0,C 180,E1 -19275.141,E2 -19275.141} C_VEL
LIN {X 0,Y 242.074,Z 441.323,A -85,B 0,C 180,E1 -19278.624,E2 -19278.624} C_VEL
LIN {X 0,Y 242.014,Z 441.311,A -85,B 0,C 180,E1 -19282.18,E2 -19282.18} C_VEL
LIN {X 0,Y 242.067,Z 441.325,A -85,B 0,C 180,E1 -19285.838,E2 -19285.838} C_VEL
LIN {X 0,Y 242.03,Z 441.336,A -85,B 0,C 180,E1 -19289.581,E2 -19289.581} C_VEL
LIN {X 0,Y 241.992,Z 441.32,A -85,B 0,C 180,E1 -19293.491,E2 -19293.491} C_VEL
LIN {X 0,Y 242.003,Z 441.34,A -85,B 0,C 180,E1 -19297.58,E2 -19297.58} C_VEL
LIN {X 0,Y 241.944,Z 441.348,A -85,B 0,C 180,E1 -19301.922,E2 -19301.922} C_VEL
LIN {X 0,Y 241.936,Z 441.344,A -85,B 0,C 180,E1 -19306.572,E2 -19306.572} C_VEL
LIN {X 0,Y 241.974,Z 441.339,A -85,B 0,C 180,E1 -19310.285,E2 -19310.285} C_VEL
LIN {X 0,Y 242.039,Z 441.328,A -85,B 0,C 180,E1 -19314.498,E2 -19314.498} C_VEL
LIN {X 0,Y 241.98,Z 441.341,A -85,B 0,C 180,E1 -19318.481,E2 -19318.481} C_VEL
LIN {X 0,Y 242.015,Z 441.334,A -85,B 0,C 180,E1 -19322.314,E2 -19322.314} C_VEL
LIN {X 0,Y 242.127,Z 441.491,A -85,B 0,C 180,E1 -19324.774,E2 -19324.774} C_VEL
LIN {X 0,Y 243.628,Z 445.385,A -85,B 0,C 180,E1 -19325.324,E2 -19325.324} C_VEL
LIN {X 0,Y 247.995,Z 456.445,A -85,B 0,C 180,E1 -19327.076,E2 -19327.076} C_VEL
LIN {X 0,Y 250.946,Z 465.343,A -85,B 0,C 180,E1 -19328.649,E2 -19328.649} C_VEL
LIN {X 0,Y 253.326,Z 475.139,A -85,B 0,C 180,E1 -19330.555,E2 -19330.555} C_VEL
LIN {X 0,Y 251.747,Z 483.827,A -85,B 0,C 180,E1 -19332.117,E2 -19332.117} C_VEL
LIN {X 0,Y 249.834,Z 492.769,A -85,B 0,C 180,E1 -19334.082,E2 -19334.082} C_VEL
LIN {X 0,Y 247.954,Z 501.45,A -85,B 0,C 180,E1 -19336.477,E2 -19336.477} C_VEL
LIN {X 0,Y 246.34,Z 508.429,A -85,B 0,C 180,E1 -19338.897,E2 -19338.897} C_VEL
LIN {X 0,Y 245.34,Z 513.114,A -85,B 0,C 180,E1 -19340.935,E2 -19340.935} C_VEL
LIN {X 0,Y 244.18,Z 517.697,A -85,B 0,C 180,E1 -19343.389,E2 -19343.389} C_VEL
LIN {X 0,Y 243.543,Z 520.164,A -85,B 0,C 180,E1 -19345.034,E2 -19345.034} C_VEL
LIN {X 0,Y 242.735,Z 523.724,A -85,B 0,C 180,E1 -19348.341,E2 -19348.341} C_VEL
LIN {X 0,Y 242.596,Z 524.904,A -85,B 0,C 180,E1 -19350,E2 -19350} C_VEL
LIN {X 0,Y 242.588,Z 525.662,A -85,B 0,C 180,E1 -19351.661,E2 -19351.661} C_VEL
LIN {X 0,Y 242.464,Z 526.092,A -85,B 0,C 180,E1 -19354.989,E2 -19354.989} C_VEL
LIN {X 0,Y 242.797,Z 525.72,A -85,B 0,C 180,E1 -19356.649,E2 -19356.649} C_VEL
LIN {X 0,Y 243.334,Z 524.928,A -85,B 0,C 180,E1 -19358.304,E2 -19358.304} C_VEL
LIN {X 0,Y 244.013,Z 523.724,A -85,B 0,C 180,E1 -19359.952,E2 -19359.952} C_VEL
LIN {X 0,Y 245.217,Z 520.527,A -85,B 0,C 180,E1 -19362.977,E2 -19362.977} C_VEL
LIN {X 0,Y 246.705,Z 516.327,A -85,B 0,C 180,E1 -19365.702,E2 -19365.702} C_VEL
LIN {X 0,Y 248.208,Z 511.351,A -85,B 0,C 180,E1 -19368.148,E2 -19368.148} C_VEL
LIN {X 0,Y 250.013,Z 505.047,A -85,B 0,C 180,E1 -19370.572,E2 -19370.572} C_VEL
LIN {X 0,Y 252.291,Z 497.143,A -85,B 0,C 180,E1 -19372.955,E2 -19372.955} C_VEL
LIN {X 0,Y 254.347,Z 489.053,A -85,B 0,C 180,E1 -19374.922,E2 -19374.922} C_VEL
LIN {X 0,Y 255.906,Z 481.734,A -85,B 0,C 180,E1 -19376.409,E2 -19376.409} C_VEL
LIN {X 0,Y 255.84,Z 478.908,A -85,B 0,C 180,E1 -19377.011,E2 -19377.011} C_VEL
LIN {X 0,Y 253.368,Z 469.317,A -85,B 0,C 180,E1 -19379.117,E2 -19379.117} C_VEL
LIN {X 0,Y 250.364,Z 460.544,A -85,B 0,C 180,E1 -19380.894,E2 -19380.894} C_VEL
LIN {X 0,Y 246.368,Z 450.995,A -85,B 0,C 180,E1 -19382.699,E2 -19382.699} C_VEL
LIN {X 0,Y 242.176,Z 442.153,A -85,B 0,C 180,E1 -19384.256,E2 -19384.256} C_VEL
LIN {X 0,Y 242.031,Z 441.338,A -85,B 0,C 180,E1 -19384.37,E2 -19384.37} C_VEL
LIN {X 0,Y 242.011,Z 441.34,A -85,B 0,C 180,E1 -19388.363,E2 -19388.363} C_VEL
LIN {X 0,Y 241.946,Z 441.348,A -85,B 0,C 180,E1 -19391.921,E2 -19391.921} C_VEL
LIN {X 0,Y 241.938,Z 441.345,A -85,B 0,C 180,E1 -19396.571,E2 -19396.571} C_VEL
LIN {X 0,Y 241.976,Z 441.339,A -85,B 0,C 180,E1 -19400.284,E2 -19400.284} C_VEL
LIN {X 0,Y 242.04,Z 441.332,A -85,B 0,C 180,E1 -19404.498,E2 -19404.498} C_VEL
LIN {X 0,Y 241.98,Z 441.341,A -85,B 0,C 180,E1 -19408.48,E2 -19408.48} C_VEL
LIN {X 0,Y 242.011,Z 441.337,A -85,B 0,C 180,E1 -19412.313,E2 -19412.313} C_VEL
LIN {X 0,Y 242.045,Z 441.332,A -85,B 0,C 180,E1 -19416.014,E2 -19416.014} C_VEL
LIN {X 0,Y 242.193,Z 441.348,A -85,B 0,C 180,E1 -19420.313,E2 -19420.313} C_VEL
LIN {X 0,Y 244.913,Z 453.741,A -85,B 0,C 180,E1 -19421.816,E2 -19421.816} C_VEL
LIN {X 0,Y 246.217,Z 459.065,A -85,B 0,C 180,E1 -19422.559,E2 -19422.559} C_VEL
LIN {X 0,Y 245.441,Z 471.285,A -85,B 0,C 180,E1 -19424.428,E2 -19424.428} C_VEL
LIN {X 0,Y 244.353,Z 482.368,A -85,B 0,C 180,E1 -19426.485,E2 -19426.485} C_VEL
LIN {X 0,Y 243.542,Z 492.124,A -85,B 0,C 180,E1 -19428.687,E2 -19428.687} C_VEL
LIN {X 0,Y 242.768,Z 501.569,A -85,B 0,C 180,E1 -19431.258,E2 -19431.258} C_VEL
LIN {X 0,Y 242.207,Z 509.061,A -85,B 0,C 180,E1 -19433.753,E2 -19433.753} C_VEL
LIN {X 0,Y 241.876,Z 514.281,A -85,B 0,C 180,E1 -19435.834,E2 -19435.834} C_VEL
LIN {X 0,Y 241.947,Z 519.487,A -85,B 0,C 180,E1 -19438.335,E2 -19438.335} C_VEL
LIN {X 0,Y 242.408,Z 523.639,A -85,B 0,C 180,E1 -19440.83,E2 -19440.83} C_VEL
LIN {X 0,Y 242.901,Z 526.851,A -85,B 0,C 180,E1 -19443.317,E2 -19443.317} C_VEL
LIN {X 0,Y 244.053,Z 529.708,A -85,B 0,C 180,E1 -19446.614,E2 -19446.614} C_VEL
LIN {X 0,Y 244.915,Z 530.587,A -85,B 0,C 180,E1 -19448.249,E2 -19448.249} C_VEL
LIN {X 0,Y 246.028,Z 531.062,A -85,B 0,C 180,E1 -19449.869,E2 -19449.869} C_VEL
LIN {X 0,Y 248.666,Z 530.847,A -85,B 0,C 180,E1 -19453.068,E2 -19453.068} C_VEL
LIN {X 0,Y 250.128,Z 530.237,A -85,B 0,C 180,E1 -19454.648,E2 -19454.648} C_VEL
LIN {X 0,Y 251.883,Z 529.211,A -85,B 0,C 180,E1 -19456.201,E2 -19456.201} C_VEL
LIN {X 0,Y 255.774,Z 526.013,A -85,B 0,C 180,E1 -19459.252,E2 -19459.252} C_VEL
LIN {X 0,Y 259.11,Z 522.583,A -85,B 0,C 180,E1 -19461.479,E2 -19461.479} C_VEL
LIN {X 0,Y 262.818,Z 518.171,A -85,B 0,C 180,E1 -19463.648,E2 -19463.648} C_VEL
LIN {X 0,Y 267.614,Z 511.707,A -85,B 0,C 180,E1 -19466.096,E2 -19466.096} C_VEL
LIN {X 0,Y 272.848,Z 503.625,A -85,B 0,C 180,E1 -19468.459,E2 -19468.459} C_VEL
LIN {X 0,Y 273.771,Z 502.042,A -85,B 0,C 180,E1 -19468.857,E2 -19468.857} C_VEL
LIN {X 0,Y 274.218,Z 499.768,A -85,B 0,C 180,E1 -19469.846,E2 -19469.846} C_VEL
LIN {X 0,Y 274.531,Z 494.608,A -85,B 0,C 180,E1 -19472.52,E2 -19472.52} C_VEL
LIN {X 0,Y 274.331,Z 490.886,A -85,B 0,C 180,E1 -19474.935,E2 -19474.935} C_VEL
LIN {X 0,Y 273.551,Z 489.002,A -85,B 0,C 180,E1 -19477.207,E2 -19477.207} C_VEL
LIN {X 0,Y 272.787,Z 488.297,A -85,B 0,C 180,E1 -19479.383,E2 -19479.383} C_VEL
LIN {X 0,Y 272.506,Z 488.429,A -85,B 0,C 180,E1 -19480.159,E2 -19480.159} C_VEL
LIN {X 0,Y 271.609,Z 489.672,A -85,B 0,C 180,E1 -19481.358,E2 -19481.358} C_VEL
LIN {X 0,Y 270.28,Z 491.908,A -85,B 0,C 180,E1 -19482.489,E2 -19482.489} C_VEL
LIN {X 0,Y 266.685,Z 499.584,A -85,B 0,C 180,E1 -19485.422,E2 -19485.422} C_VEL
LIN {X 0,Y 266.215,Z 501.263,A -85,B 0,C 180,E1 -19486.206,E2 -19486.206} C_VEL
LIN {X 0,Y 265.715,Z 503.686,A -85,B 0,C 180,E1 -19487.307,E2 -19487.307} C_VEL
LIN {X 0,Y 263.09,Z 512.63,A -85,B 0,C 180,E1 -19490.124,E2 -19490.124} C_VEL
LIN {X 0,Y 260.016,Z 524.497,A -85,B 0,C 180,E1 -19493.512,E2 -19493.512} C_VEL
LIN {X 0,Y 256.808,Z 535.49,A -85,B 0,C 180,E1 -19496.467,E2 -19496.467} C_VEL
LIN {X 0,Y 253.219,Z 546.098,A -85,B 0,C 180,E1 -19499.361,E2 -19499.361} C_VEL
LIN {X 0,Y 248.125,Z 557.304,A -85,B 0,C 180,E1 -19502.595,E2 -19502.595} C_VEL
LIN {X 0,Y 243.766,Z 566.263,A -85,B 0,C 180,E1 -19505.742,E2 -19505.742} C_VEL
LIN {X 0,Y 240.019,Z 572.841,A -85,B 0,C 180,E1 -19508.53,E2 -19508.53} C_VEL
LIN {X 0,Y 236.782,Z 578.818,A -85,B 0,C 180,E1 -19511.769,E2 -19511.769} C_VEL
LIN {X 0,Y 235.142,Z 582.507,A -85,B 0,C 180,E1 -19514.395,E2 -19514.395} C_VEL
LIN {X 0,Y 233.804,Z 587.02,A -85,B 0,C 180,E1 -19518.732,E2 -19518.732} C_VEL
LIN {X 0,Y 233.728,Z 590.426,A -85,B 0,C 180,E1 -19521.353,E2 -19521.353} C_VEL
LIN {X 0,Y 233.877,Z 592.162,A -85,B 0,C 180,E1 -19523.096,E2 -19523.096} C_VEL
LIN {X 0,Y 234.146,Z 593.468,A -85,B 0,C 180,E1 -19524.833,E2 -19524.833} C_VEL
LIN {X 0,Y 234.806,Z 594.768,A -85,B 0,C 180,E1 -19528.284,E2 -19528.284} C_VEL
LIN {X 0,Y 235.358,Z 594.834,A -85,B 0,C 180,E1 -19530,E2 -19530} C_VEL
LIN {X 0,Y 234.824,Z 594.318,A -85,B 0,C 180,E1 -19531.715,E2 -19531.715} C_VEL
LIN {X 0,Y 234.477,Z 593.363,A -85,B 0,C 180,E1 -19533.436,E2 -19533.436} C_VEL
LIN {X 0,Y 234.232,Z 591.998,A -85,B 0,C 180,E1 -19535.164,E2 -19535.164} C_VEL
LIN {X 0,Y 233.932,Z 589.441,A -85,B 0,C 180,E1 -19537.513,E2 -19537.513} C_VEL
LIN {X 0,Y 233.83,Z 585.149,A -85,B 0,C 180,E1 -19540.389,E2 -19540.389} C_VEL
LIN {X 0,Y 234.245,Z 580.07,A -85,B 0,C 180,E1 -19543.004,E2 -19543.004} C_VEL
LIN {X 0,Y 235.07,Z 573.706,A -85,B 0,C 180,E1 -19545.609,E2 -19545.609} C_VEL
LIN {X 0,Y 236.361,Z 567.227,A -85,B 0,C 180,E1 -19547.763,E2 -19547.763} C_VEL
LIN {X 0,Y 238.335,Z 557.925,A -85,B 0,C 180,E1 -19550.272,E2 -19550.272} C_VEL
LIN {X 0,Y 239.372,Z 548.042,A -85,B 0,C 180,E1 -19552.438,E2 -19552.438} C_VEL
LIN {X 0,Y 240.115,Z 537.125,A -85,B 0,C 180,E1 -19554.406,E2 -19554.406} C_VEL
LIN {X 0,Y 240.369,Z 526.375,A -85,B 0,C 180,E1 -19556.013,E2 -19556.013} C_VEL
LIN {X 0,Y 240.058,Z 515.101,A -85,B 0,C 180,E1 -19557.421,E2 -19557.421} C_VEL
LIN {X 0,Y 239.09,Z 502.757,A -85,B 0,C 180,E1 -19558.689,E2 -19558.689} C_VEL
LIN {X 0,Y 237.191,Z 489.33,A -85,B 0,C 180,E1 -19559.803,E2 -19559.803} C_VEL
LIN {X 0,Y 235.973,Z 482.247,A -85,B 0,C 180,E1 -19560.325,E2 -19560.325} C_VEL
LIN {X 0,Y 237.77,Z 473.065,A -85,B 0,C 180,E1 -19565.196,E2 -19565.196} C_VEL
LIN {X 0,Y 239.259,Z 465.679,A -85,B 0,C 180,E1 -19569.116,E2 -19569.116} C_VEL
LIN {X 0,Y 238.787,Z 461.764,A -85,B 0,C 180,E1 -19571.417,E2 -19571.417} C_VEL
LIN {X 0,Y 237.6,Z 455.53,A -85,B 0,C 180,E1 -19575.226,E2 -19575.226} C_VEL
LIN {X 0,Y 236.41,Z 449.458,A -85,B 0,C 180,E1 -19579.155,E2 -19579.155} C_VEL
LIN {X 0,Y 235.093,Z 442.84,A -85,B 0,C 180,E1 -19583.818,E2 -19583.818} C_VEL
LIN {X 0,Y 234.98,Z 442.216,A -85,B 0,C 180,E1 -19584.297,E2 -19584.297} C_VEL
LIN {X 0,Y 234.96,Z 442.219,A -85,B 0,C 180,E1 -19587.425,E2 -19587.425} C_VEL
LIN {X 0,Y 234.937,Z 442.221,A -85,B 0,C 180,E1 -19591.404,E2 -19591.404} C_VEL
LIN {X 0,Y 234.989,Z 442.213,A -85,B 0,C 180,E1 -19595.247,E2 -19595.247} C_VEL
LIN {X 0,Y 235.028,Z 442.21,A -85,B 0,C 180,E1 -19598.972,E2 -19598.972} C_VEL
LIN {X 0,Y 235.097,Z 442.202,A -85,B 0,C 180,E1 -19603.059,E2 -19603.059} C_VEL
LIN {X 0,Y 235.116,Z 442.2,A -85,B 0,C 180,E1 -19607.922,E2 -19607.922} C_VEL
LIN {X 0,Y 235.327,Z 442.172,A -85,B 0,C 180,E1 -19611.412,E2 -19611.412} C_VEL
LIN {X 0,Y 235.369,Z 442.165,A -85,B 0,C 180,E1 -19613.141,E2 -19613.141} C_VEL
LIN {X 0,Y 235.598,Z 442.138,A -85,B 0,C 180,E1 -19618.291,E2 -19618.291} C_VEL
LIN {X 0,Y 235.597,Z 442.137,A -85,B 0,C 180,E1 -19621.71,E2 -19621.71} C_VEL
LIN {X 0,Y 235.407,Z 442.154,A -85,B 0,C 180,E1 -19626.859,E2 -19626.859} C_VEL
LIN {X 0,Y 235.254,Z 442.179,A -85,B 0,C 180,E1 -19630.326,E2 -19630.326} C_VEL
LIN {X 0,Y 235.115,Z 442.196,A -85,B 0,C 180,E1 -19635.607,E2 -19635.607} C_VEL
LIN {X 0,Y 235.01,Z 442.202,A -85,B 0,C 180,E1 -19639.206,E2 -19639.206} C_VEL
LIN {X 0,Y 234.962,Z 442.189,A -85,B 0,C 180,E1 -19642.883,E2 -19642.883} C_VEL
LIN {X 0,Y 234.97,Z 442.213,A -85,B 0,C 180,E1 -19646.658,E2 -19646.658} C_VEL
LIN {X 0,Y 234.933,Z 442.212,A -85,B 0,C 180,E1 -19650.568,E2 -19650.568} C_VEL
LIN {X 0,Y 234.962,Z 442.203,A -85,B 0,C 180,E1 -19654.633,E2 -19654.633} C_VEL
LIN {X 0,Y 234.943,Z 442.217,A -85,B 0,C 180,E1 -19658.945,E2 -19658.945} C_VEL
LIN {X 0,Y 234.888,Z 442.224,A -85,B 0,C 180,E1 -19663.486,E2 -19663.486} C_VEL
LIN {X 0,Y 234.889,Z 442.222,A -85,B 0,C 180,E1 -19666.515,E2 -19666.515} C_VEL
LIN {X 0,Y 234.957,Z 442.212,A -85,B 0,C 180,E1 -19671.087,E2 -19671.087} C_VEL
LIN {X 0,Y 234.963,Z 442.211,A -85,B 0,C 180,E1 -19675.368,E2 -19675.368} C_VEL
LIN {X 0,Y 234.973,Z 442.209,A -85,B 0,C 180,E1 -19680.157,E2 -19680.157} C_VEL
LIN {X 0,Y 235.021,Z 442.209,A -85,B 0,C 180,E1 -19683.851,E2 -19683.851} C_VEL
LIN {X 0,Y 235.735,Z 444.485,A -85,B 0,C 180,E1 -19684.164,E2 -19684.164} C_VEL
LIN {X 0,Y 239.353,Z 452.997,A -85,B 0,C 180,E1 -19685.539,E2 -19685.539} C_VEL
LIN {X 0,Y 242.931,Z 462.786,A -85,B 0,C 180,E1 -19687.276,E2 -19687.276} C_VEL
LIN {X 0,Y 245.746,Z 472.671,A -85,B 0,C 180,E1 -19689.21,E2 -19689.21} C_VEL
LIN {X 0,Y 246.65,Z 476.928,A -85,B 0,C 180,E1 -19690.103,E2 -19690.103} C_VEL
LIN {X 0,Y 244.7,Z 486.971,A -85,B 0,C 180,E1 -19692.016,E2 -19692.016} C_VEL
LIN {X 0,Y 242.775,Z 495.552,A -85,B 0,C 180,E1 -19694.038,E2 -19694.038} C_VEL
LIN {X 0,Y 240.832,Z 503.882,A -85,B 0,C 180,E1 -19696.5,E2 -19696.5} C_VEL
LIN {X 0,Y 239.258,Z 510.538,A -85,B 0,C 180,E1 -19698.993,E2 -19698.993} C_VEL
LIN {X 0,Y 238.009,Z 515.857,A -85,B 0,C 180,E1 -19701.51,E2 -19701.51} C_VEL
LIN {X 0,Y 236.873,Z 520.052,A -85,B 0,C 180,E1 -19704.04,E2 -19704.04} C_VEL
LIN {X 0,Y 236.033,Z 523.213,A -85,B 0,C 180,E1 -19706.586,E2 -19706.586} C_VEL
LIN {X 0,Y 235.571,Z 525.946,A -85,B 0,C 180,E1 -19710,E2 -19710} C_VEL
LIN {X 0,Y 235.563,Z 526.688,A -85,B 0,C 180,E1 -19711.71,E2 -19711.71} C_VEL
LIN {X 0,Y 235.456,Z 527.101,A -85,B 0,C 180,E1 -19715.138,E2 -19715.138} C_VEL
LIN {X 0,Y 235.812,Z 526.719,A -85,B 0,C 180,E1 -19716.847,E2 -19716.847} C_VEL
LIN {X 0,Y 236.379,Z 525.907,A -85,B 0,C 180,E1 -19718.55,E2 -19718.55} C_VEL
LIN {X 0,Y 237.091,Z 524.694,A -85,B 0,C 180,E1 -19720.245,E2 -19720.245} C_VEL
LIN {X 0,Y 238.371,Z 521.481,A -85,B 0,C 180,E1 -19723.353,E2 -19723.353} C_VEL
LIN {X 0,Y 239.931,Z 517.254,A -85,B 0,C 180,E1 -19726.158,E2 -19726.158} C_VEL
LIN {X 0,Y 241.524,Z 512.251,A -85,B 0,C 180,E1 -19728.668,E2 -19728.668} C_VEL
LIN {X 0,Y 243.431,Z 505.919,A -85,B 0,C 180,E1 -19731.155,E2 -19731.155} C_VEL
LIN {X 0,Y 245.823,Z 497.986,A -85,B 0,C 180,E1 -19733.595,E2 -19733.595} C_VEL
LIN {X 0,Y 247.981,Z 489.86,A -85,B 0,C 180,E1 -19735.608,E2 -19735.608} C_VEL
LIN {X 0,Y 249.506,Z 482.729,A -85,B 0,C 180,E1 -19737.094,E2 -19737.094} C_VEL
LIN {X 0,Y 248.035,Z 475.523,A -85,B 0,C 180,E1 -19738.796,E2 -19738.796} C_VEL
LIN {X 0,Y 245.372,Z 466.581,A -85,B 0,C 180,E1 -19740.765,E2 -19740.765} C_VEL
LIN {X 0,Y 241.949,Z 457.672,A -85,B 0,C 180,E1 -19742.607,E2 -19742.607} C_VEL
LIN {X 0,Y 237.031,Z 446.879,A -85,B 0,C 180,E1 -19744.686,E2 -19744.686} C_VEL
LIN {X 0,Y 235.192,Z 443.22,A -85,B 0,C 180,E1 -19745.363,E2 -19745.363} C_VEL
LIN {X 0,Y 235.008,Z 442.211,A -85,B 0,C 180,E1 -19745.523,E2 -19745.523} C_VEL
LIN {X 0,Y 234.945,Z 442.218,A -85,B 0,C 180,E1 -19748.944,E2 -19748.944} C_VEL
LIN {X 0,Y 234.891,Z 442.224,A -85,B 0,C 180,E1 -19753.486,E2 -19753.486} C_VEL
LIN {X 0,Y 234.891,Z 442.223,A -85,B 0,C 180,E1 -19756.514,E2 -19756.514} C_VEL
LIN {X 0,Y 234.958,Z 442.213,A -85,B 0,C 180,E1 -19761.086,E2 -19761.086} C_VEL
LIN {X 0,Y 234.964,Z 442.214,A -85,B 0,C 180,E1 -19765.367,E2 -19765.367} C_VEL
LIN {X 0,Y 234.973,Z 442.215,A -85,B 0,C 180,E1 -19770.157,E2 -19770.157} C_VEL
LIN {X 0,Y 234.998,Z 442.214,A -85,B 0,C 180,E1 -19773.794,E2 -19773.794} C_VEL
LIN {X 0,Y 235.029,Z 442.207,A -85,B 0,C 180,E1 -19778.971,E2 -19778.971} C_VEL
LIN {X 0,Y 235.146,Z 442.384,A -85,B 0,C 180,E1 -19780.181,E2 -19780.181} C_VEL
LIN {X 0,Y 238.284,Z 456.48,A -85,B 0,C 180,E1 -19781.966,E2 -19781.966} C_VEL
LIN {X 0,Y 239.198,Z 460.56,A -85,B 0,C 180,E1 -19782.563,E2 -19782.563} C_VEL
LIN {X 0,Y 238.147,Z 473.355,A -85,B 0,C 180,E1 -19784.597,E2 -19784.597} C_VEL
LIN {X 0,Y 237.117,Z 484.289,A -85,B 0,C 180,E1 -19786.72,E2 -19786.72} C_VEL
LIN {X 0,Y 236.273,Z 494.284,A -85,B 0,C 180,E1 -19789.09,E2 -19789.09} C_VEL
LIN {X 0,Y 235.627,Z 502.474,A -85,B 0,C 180,E1 -19791.423,E2 -19791.423} C_VEL
LIN {X 0,Y 235.081,Z 510.009,A -85,B 0,C 180,E1 -19793.993,E2 -19793.993} C_VEL
LIN {X 0,Y 234.823,Z 516.217,A -85,B 0,C 180,E1 -19796.568,E2 -19796.568} C_VEL
LIN {X 0,Y 235.029,Z 521.302,A -85,B 0,C 180,E1 -19799.143,E2 -19799.143} C_VEL
LIN {X 0,Y 235.449,Z 525.331,A -85,B 0,C 180,E1 -19801.71,E2 -19801.71} C_VEL
LIN {X 0,Y 236.381,Z 529.296,A -85,B 0,C 180,E1 -19805.117,E2 -19805.117} C_VEL
LIN {X 0,Y 237.981,Z 531.683,A -85,B 0,C 180,E1 -19808.491,E2 -19808.491} C_VEL
LIN {X 0,Y 240.47,Z 532.552,A -85,B 0,C 180,E1 -19811.805,E2 -19811.805} C_VEL
LIN {X 0,Y 243.473,Z 531.925,A -85,B 0,C 180,E1 -19815.057,E2 -19815.057} C_VEL
LIN {X 0,Y 247.275,Z 529.865,A -85,B 0,C 180,E1 -19818.218,E2 -19818.218} C_VEL
LIN {X 0,Y 251.713,Z 526.219,A -85,B 0,C 180,E1 -19821.282,E2 -19821.282} C_VEL
LIN {X 0,Y 255.497,Z 522.471,A -85,B 0,C 180,E1 -19823.506,E2 -19823.506} C_VEL
LIN {X 0,Y 261.071,Z 515.95,A -85,B 0,C 180,E1 -19826.371,E2 -19826.371} C_VEL
LIN {X 0,Y 266.464,Z 508.604,A -85,B 0,C 180,E1 -19828.773,E2 -19828.773} C_VEL
LIN {X 0,Y 268.802,Z 505.073,A -85,B 0,C 180,E1 -19829.786,E2 -19829.786} C_VEL
LIN {X 0,Y 269.605,Z 500.368,A -85,B 0,C 180,E1 -19832.347,E2 -19832.347} C_VEL
LIN {X 0,Y 269.823,Z 496.546,A -85,B 0,C 180,E1 -19834.962,E2 -19834.962} C_VEL
LIN {X 0,Y 269.457,Z 494.976,A -85,B 0,C 180,E1 -19836.862,E2 -19836.862} C_VEL
LIN {X 0,Y 268.946,Z 494.25,A -85,B 0,C 180,E1 -19838.841,E2 -19838.841} C_VEL
LIN {X 0,Y 268.192,Z 494.704,A -85,B 0,C 180,E1 -19840.929,E2 -19840.929} C_VEL
LIN {X 0,Y 267.375,Z 496.518,A -85,B 0,C 180,E1 -19843.111,E2 -19843.111} C_VEL
LIN {X 0,Y 266.33,Z 500.687,A -85,B 0,C 180,E1 -19845.904,E2 -19845.904} C_VEL
LIN {X 0,Y 266.215,Z 501.263,A -85,B 0,C 180,E1 -19846.206,E2 -19846.206} C_VEL
LIN {X 0,Y 265.678,Z 503.134,A -85,B 0,C 180,E1 -19846.944,E2 -19846.944} C_VEL
LIN {X 0,Y 264.7,Z 505.546,A -85,B 0,C 180,E1 -19847.588,E2 -19847.588} C_VEL
LIN {X 0,Y 261.907,Z 511.161,A -85,B 0,C 180,E1 -19848.69,E2 -19848.69} C_VEL
LIN {X 0,Y 258.869,Z 516.897,A -85,B 0,C 180,E1 -19849.758,E2 -19849.758} C_VEL
LIN {X 0,Y 257.019,Z 520.861,A -85,B 0,C 180,E1 -19850.68,E2 -19850.68} C_VEL
LIN {X 0,Y 256.583,Z 522.056,A -85,B 0,C 180,E1 -19851.027,E2 -19851.027} C_VEL
LIN {X 0,Y 253.29,Z 531.989,A -85,B 0,C 180,E1 -19853.969,E2 -19853.969} C_VEL
LIN {X 0,Y 248.717,Z 544.251,A -85,B 0,C 180,E1 -19857.528,E2 -19857.528} C_VEL
LIN {X 0,Y 245.714,Z 550.88,A -85,B 0,C 180,E1 -19859.501,E2 -19859.501} C_VEL
LIN {X 0,Y 240.675,Z 560.425,A -85,B 0,C 180,E1 -19862.618,E2 -19862.618} C_VEL
LIN {X 0,Y 236.749,Z 567.587,A -85,B 0,C 180,E1 -19865.443,E2 -19865.443} C_VEL
LIN {X 0,Y 232.462,Z 574.381,A -85,B 0,C 180,E1 -19868.728,E2 -19868.728} C_VEL
LIN {X 0,Y 229.325,Z 579.723,A -85,B 0,C 180,E1 -19872.153,E2 -19872.153} C_VEL
LIN {X 0,Y 227.493,Z 583.663,A -85,B 0,C 180,E1 -19875.691,E2 -19875.691} C_VEL
LIN {X 0,Y 226.805,Z 586.051,A -85,B 0,C 180,E1 -19878.38,E2 -19878.38} C_VEL
LIN {X 0,Y 226.656,Z 589.438,A -85,B 0,C 180,E1 -19881.081,E2 -19881.081} C_VEL
LIN {X 0,Y 226.782,Z 591.167,A -85,B 0,C 180,E1 -19882.879,E2 -19882.879} C_VEL
LIN {X 0,Y 227.058,Z 592.462,A -85,B 0,C 180,E1 -19884.672,E2 -19884.672} C_VEL
LIN {X 0,Y 227.349,Z 593.306,A -85,B 0,C 180,E1 -19886.455,E2 -19886.455} C_VEL
LIN {X 0,Y 228.319,Z 593.816,A -85,B 0,C 180,E1 -19890,E2 -19890} C_VEL
LIN {X 0,Y 227.759,Z 593.282,A -85,B 0,C 180,E1 -19891.768,E2 -19891.768} C_VEL
LIN {X 0,Y 227.415,Z 592.318,A -85,B 0,C 180,E1 -19893.543,E2 -19893.543} C_VEL
LIN {X 0,Y 227.143,Z 590.938,A -85,B 0,C 180,E1 -19895.326,E2 -19895.326} C_VEL
LIN {X 0,Y 226.86,Z 588.618,A -85,B 0,C 180,E1 -19897.545,E2 -19897.545} C_VEL
LIN {X 0,Y 226.773,Z 584.046,A -85,B 0,C 180,E1 -19900.716,E2 -19900.716} C_VEL
LIN {X 0,Y 227.269,Z 578.951,A -85,B 0,C 180,E1 -19903.41,E2 -19903.41} C_VEL
LIN {X 0,Y 228.164,Z 572.565,A -85,B 0,C 180,E1 -19906.094,E2 -19906.094} C_VEL
LIN {X 0,Y 229.768,Z 565.381,A -85,B 0,C 180,E1 -19908.521,E2 -19908.521} C_VEL
LIN {X 0,Y 231.569,Z 556.712,A -85,B 0,C 180,E1 -19910.892,E2 -19910.892} C_VEL
LIN {X 0,Y 232.555,Z 546.761,A -85,B 0,C 180,E1 -19913.133,E2 -19913.133} C_VEL
LIN {X 0,Y 233.336,Z 536.065,A -85,B 0,C 180,E1 -19915.114,E2 -19915.114} C_VEL
LIN {X 0,Y 233.643,Z 524.966,A -85,B 0,C 180,E1 -19916.82,E2 -19916.82} C_VEL
LIN {X 0,Y 233.378,Z 514.195,A -85,B 0,C 180,E1 -19918.205,E2 -19918.205} C_VEL
LIN {X 0,Y 232.281,Z 501.071,A -85,B 0,C 180,E1 -19919.605,E2 -19919.605} C_VEL
LIN {X 0,Y 230.298,Z 487.637,A -85,B 0,C 180,E1 -19920.765,E2 -19920.765} C_VEL
LIN {X 0,Y 229.172,Z 481.182,A -85,B 0,C 180,E1 -19921.264,E2 -19921.264} C_VEL
LIN {X 0,Y 230.725,Z 473.725,A -85,B 0,C 180,E1 -19925.362,E2 -19925.362} C_VEL
LIN {X 0,Y 232.06,Z 467.746,A -85,B 0,C 180,E1 -19928.619,E2 -19928.619} C_VEL
LIN {X 0,Y 232.183,Z 465.211,A -85,B 0,C 180,E1 -19930.095,E2 -19930.095} C_VEL
LIN {X 0,Y 230.902,Z 458.264,A -85,B 0,C 180,E1 -19934.431,E2 -19934.431} C_VEL
LIN {X 0,Y 229.619,Z 451.6,A -85,B 0,C 180,E1 -19938.848,E2 -19938.848} C_VEL
LIN {X 0,Y 228.446,Z 445.636,A -85,B 0,C 180,E1 -19943.118,E2 -19943.118} C_VEL
LIN {X 0,Y 227.925,Z 443.096,A -85,B 0,C 180,E1 -19945.084,E2 -19945.084} C_VEL
LIN {X 0,Y 227.904,Z 443.097,A -85,B 0,C 180,E1 -19950.436,E2 -19950.436} C_VEL
LIN {X 0,Y 227.929,Z 443.094,A -85,B 0,C 180,E1 -19954.426,E2 -19954.426} C_VEL
LIN {X 0,Y 227.992,Z 443.088,A -85,B 0,C 180,E1 -19958.29,E2 -19958.29} C_VEL
LIN {X 0,Y 228.036,Z 443.082,A -85,B 0,C 180,E1 -19962.825,E2 -19962.825} C_VEL
LIN {X 0,Y 228.074,Z 443.076,A -85,B 0,C 180,E1 -19967.543,E2 -19967.543} C_VEL
LIN {X 0,Y 228.264,Z 443.052,A -85,B 0,C 180,E1 -19971.145,E2 -19971.145} C_VEL
LIN {X 0,Y 228.32,Z 443.044,A -85,B 0,C 180,E1 -19972.928,E2 -19972.928} C_VEL
LIN {X 0,Y 228.556,Z 443.015,A -85,B 0,C 180,E1 -19978.238,E2 -19978.238} C_VEL
LIN {X 0,Y 228.556,Z 443.014,A -85,B 0,C 180,E1 -19981.762,E2 -19981.762} C_VEL
LIN {X 0,Y 228.359,Z 443.032,A -85,B 0,C 180,E1 -19987.072,E2 -19987.072} C_VEL
LIN {X 0,Y 228.168,Z 443.06,A -85,B 0,C 180,E1 -19990.65,E2 -19990.65} C_VEL
LIN {X 0,Y 228.066,Z 443.072,A -85,B 0,C 180,E1 -19994.272,E2 -19994.272} C_VEL
LIN {X 0,Y 228.004,Z 443.079,A -85,B 0,C 180,E1 -19997.954,E2 -19997.954} C_VEL
LIN {X 0,Y 227.931,Z 443.062,A -85,B 0,C 180,E1 -20002.33,E2 -20002.33} C_VEL
LIN {X 0,Y 227.944,Z 443.089,A -85,B 0,C 180,E1 -20006.603,E2 -20006.603} C_VEL
LIN {X 0,Y 227.909,Z 443.088,A -85,B 0,C 180,E1 -20010.296,E2 -20010.296} C_VEL
LIN {X 0,Y 227.89,Z 443.074,A -85,B 0,C 180,E1 -20013.719,E2 -20013.719} C_VEL
LIN {X 0,Y 227.871,Z 443.101,A -85,B 0,C 180,E1 -20018.086,E2 -20018.086} C_VEL
LIN {X 0,Y 227.815,Z 443.104,A -85,B 0,C 180,E1 -20022.742,E2 -20022.742} C_VEL
LIN {X 0,Y 227.816,Z 443.103,A -85,B 0,C 180,E1 -20027.259,E2 -20027.259} C_VEL
LIN {X 0,Y 227.872,Z 443.094,A -85,B 0,C 180,E1 -20031.915,E2 -20031.915} C_VEL
LIN {X 0,Y 227.893,Z 443.094,A -85,B 0,C 180,E1 -20036.373,E2 -20036.373} C_VEL
LIN {X 0,Y 227.923,Z 443.085,A -85,B 0,C 180,E1 -20040.439,E2 -20040.439} C_VEL
LIN {X 0,Y 227.92,Z 443.105,A -85,B 0,C 180,E1 -20042.89,E2 -20042.89} C_VEL
LIN {X 0,Y 228.452,Z 445.017,A -85,B 0,C 180,E1 -20043.145,E2 -20043.145} C_VEL
LIN {X 0,Y 232.392,Z 453.661,A -85,B 0,C 180,E1 -20044.641,E2 -20044.641} C_VEL
LIN {X 0,Y 236.112,Z 463.976,A -85,B 0,C 180,E1 -20046.54,E2 -20046.54} C_VEL
LIN {X 0,Y 238.627,Z 472.332,A -85,B 0,C 180,E1 -20048.234,E2 -20048.234} C_VEL
LIN {X 0,Y 239.995,Z 478.432,A -85,B 0,C 180,E1 -20049.569,E2 -20049.569} C_VEL
LIN {X 0,Y 238.056,Z 488.202,A -85,B 0,C 180,E1 -20051.497,E2 -20051.497} C_VEL
LIN {X 0,Y 236.059,Z 496.746,A -85,B 0,C 180,E1 -20053.571,E2 -20053.571} C_VEL
LIN {X 0,Y 234.024,Z 505.032,A -85,B 0,C 180,E1 -20056.099,E2 -20056.099} C_VEL
LIN {X 0,Y 232.381,Z 511.663,A -85,B 0,C 180,E1 -20058.663,E2 -20058.663} C_VEL
LIN {X 0,Y 231.072,Z 516.96,A -85,B 0,C 180,E1 -20061.253,E2 -20061.253} C_VEL
LIN {X 0,Y 229.889,Z 521.135,A -85,B 0,C 180,E1 -20063.858,E2 -20063.858} C_VEL
LIN {X 0,Y 229.022,Z 524.275,A -85,B 0,C 180,E1 -20066.482,E2 -20066.482} C_VEL
LIN {X 0,Y 228.545,Z 526.987,A -85,B 0,C 180,E1 -20070,E2 -20070} C_VEL
LIN {X 0,Y 228.538,Z 527.713,A -85,B 0,C 180,E1 -20071.763,E2 -20071.763} C_VEL
LIN {X 0,Y 228.451,Z 528.109,A -85,B 0,C 180,E1 -20075.296,E2 -20075.296} C_VEL
LIN {X 0,Y 228.83,Z 527.715,A -85,B 0,C 180,E1 -20077.057,E2 -20077.057} C_VEL
LIN {X 0,Y 230.176,Z 525.665,A -85,B 0,C 180,E1 -20080.557,E2 -20080.557} C_VEL
LIN {X 0,Y 231.535,Z 522.436,A -85,B 0,C 180,E1 -20083.752,E2 -20083.752} C_VEL
LIN {X 0,Y 233.15,Z 518.183,A -85,B 0,C 180,E1 -20086.641,E2 -20086.641} C_VEL
LIN {X 0,Y 234.862,Z 513.149,A -85,B 0,C 180,E1 -20089.218,E2 -20089.218} C_VEL
LIN {X 0,Y 236.876,Z 506.791,A -85,B 0,C 180,E1 -20091.77,E2 -20091.77} C_VEL
LIN {X 0,Y 239.373,Z 498.83,A -85,B 0,C 180,E1 -20094.271,E2 -20094.271} C_VEL
LIN {X 0,Y 241.651,Z 490.668,A -85,B 0,C 180,E1 -20096.329,E2 -20096.329} C_VEL
LIN {X 0,Y 242.968,Z 484.913,A -85,B 0,C 180,E1 -20097.569,E2 -20097.569} C_VEL
LIN {X 0,Y 241.959,Z 479.132,A -85,B 0,C 180,E1 -20099.001,E2 -20099.001} C_VEL
LIN {X 0,Y 239.549,Z 470.472,A -85,B 0,C 180,E1 -20101.045,E2 -20101.045} C_VEL
LIN {X 0,Y 236.182,Z 461.36,A -85,B 0,C 180,E1 -20103.067,E2 -20103.067} C_VEL
LIN {X 0,Y 231.73,Z 451.116,A -85,B 0,C 180,E1 -20105.187,E2 -20105.187} C_VEL
LIN {X 0,Y 229.641,Z 446.901,A -85,B 0,C 180,E1 -20106.027,E2 -20106.027} C_VEL
LIN {X 0,Y 228.206,Z 444.432,A -85,B 0,C 180,E1 -20106.542,E2 -20106.542} C_VEL
LIN {X 0,Y 227.916,Z 443.096,A -85,B 0,C 180,E1 -20106.756,E2 -20106.756} C_VEL
LIN {X 0,Y 227.837,Z 443.105,A -85,B 0,C 180,E1 -20110.375,E2 -20110.375} C_VEL
LIN {X 0,Y 227.837,Z 443.103,A -85,B 0,C 180,E1 -20115.193,E2 -20115.193} C_VEL
LIN {X 0,Y 227.837,Z 443.104,A -85,B 0,C 180,E1 -20119.625,E2 -20119.625} C_VEL
LIN {X 0,Y 227.903,Z 443.092,A -85,B 0,C 180,E1 -20124.132,E2 -20124.132} C_VEL
LIN {X 0,Y 227.877,Z 443.097,A -85,B 0,C 180,E1 -20128.378,E2 -20128.378} C_VEL
LIN {X 0,Y 227.89,Z 443.096,A -85,B 0,C 180,E1 -20132.445,E2 -20132.445} C_VEL
LIN {X 0,Y 227.91,Z 443.094,A -85,B 0,C 180,E1 -20136.367,E2 -20136.367} C_VEL
LIN {X 0,Y 228.067,Z 443.073,A -85,B 0,C 180,E1 -20140.009,E2 -20140.009} C_VEL
LIN {X 0,Y 231.06,Z 456.735,A -85,B 0,C 180,E1 -20141.774,E2 -20141.774} C_VEL
LIN {X 0,Y 232.01,Z 460.695,A -85,B 0,C 180,E1 -20142.367,E2 -20142.367} C_VEL
LIN {X 0,Y 231.306,Z 471.756,A -85,B 0,C 180,E1 -20144.13,E2 -20144.13} C_VEL
LIN {X 0,Y 230.071,Z 484.023,A -85,B 0,C 180,E1 -20146.531,E2 -20146.531} C_VEL
LIN {X 0,Y 229.189,Z 494.32,A -85,B 0,C 180,E1 -20148.995,E2 -20148.995} C_VEL
LIN {X 0,Y 228.479,Z 503.327,A -85,B 0,C 180,E1 -20151.598,E2 -20151.598} C_VEL
LIN {X 0,Y 227.916,Z 510.947,A -85,B 0,C 180,E1 -20154.248,E2 -20154.248} C_VEL
LIN {X 0,Y 227.733,Z 516.229,A -85,B 0,C 180,E1 -20156.461,E2 -20156.461} C_VEL
LIN {X 0,Y 227.954,Z 521.533,A -85,B 0,C 180,E1 -20159.116,E2 -20159.116} C_VEL
LIN {X 0,Y 228.369,Z 525.806,A -85,B 0,C 180,E1 -20161.763,E2 -20161.763} C_VEL
LIN {X 0,Y 229.37,Z 530.04,A -85,B 0,C 180,E1 -20165.274,E2 -20165.274} C_VEL
LIN {X 0,Y 231.049,Z 532.757,A -85,B 0,C 180,E1 -20168.748,E2 -20168.748} C_VEL
LIN {X 0,Y 233.67,Z 533.886,A -85,B 0,C 180,E1 -20172.154,E2 -20172.154} C_VEL
LIN {X 0,Y 236.842,Z 533.63,A -85,B 0,C 180,E1 -20175.489,E2 -20175.489} C_VEL
LIN {X 0,Y 240.817,Z 531.848,A -85,B 0,C 180,E1 -20178.725,E2 -20178.725} C_VEL
LIN {X 0,Y 245.501,Z 528.648,A -85,B 0,C 180,E1 -20181.848,E2 -20181.848} C_VEL
LIN {X 0,Y 250.841,Z 523.827,A -85,B 0,C 180,E1 -20184.851,E2 -20184.851} C_VEL
LIN {X 0,Y 255.301,Z 519.11,A -85,B 0,C 180,E1 -20187.014,E2 -20187.014} C_VEL
LIN {X 0,Y 260.939,Z 512.328,A -85,B 0,C 180,E1 -20189.442,E2 -20189.442} C_VEL
LIN {X 0,Y 263.503,Z 508.883,A -85,B 0,C 180,E1 -20190.448,E2 -20190.448} C_VEL
LIN {X 0,Y 264.349,Z 506.023,A -85,B 0,C 180,E1 -20192.122,E2 -20192.122} C_VEL
LIN {X 0,Y 265.069,Z 502.363,A -85,B 0,C 180,E1 -20194.721,E2 -20194.721} C_VEL
LIN {X 0,Y 265.112,Z 501.38,A -85,B 0,C 180,E1 -20195.677,E2 -20195.677} C_VEL
LIN {X 0,Y 264.876,Z 500.233,A -85,B 0,C 180,E1 -20197.608,E2 -20197.608} C_VEL
LIN {X 0,Y 264.382,Z 500.099,A -85,B 0,C 180,E1 -20199.642,E2 -20199.642} C_VEL
LIN {X 0,Y 263.585,Z 501.262,A -85,B 0,C 180,E1 -20201.804,E2 -20201.804} C_VEL
LIN {X 0,Y 263.202,Z 502.169,A -85,B 0,C 180,E1 -20202.843,E2 -20202.843} C_VEL
LIN {X 0,Y 262.242,Z 505.258,A -85,B 0,C 180,E1 -20205.032,E2 -20205.032} C_VEL
LIN {X 0,Y 261.444,Z 508.159,A -85,B 0,C 180,E1 -20206.535,E2 -20206.535} C_VEL
LIN {X 0,Y 258.497,Z 516.348,A -85,B 0,C 180,E1 -20209.268,E2 -20209.268} C_VEL
LIN {X 0,Y 256.583,Z 522.056,A -85,B 0,C 180,E1 -20211.027,E2 -20211.027} C_VEL
LIN {X 0,Y 254.962,Z 525.813,A -85,B 0,C 180,E1 -20211.997,E2 -20211.997} C_VEL
LIN {X 0,Y 250.819,Z 532.695,A -85,B 0,C 180,E1 -20213.351,E2 -20213.351} C_VEL
LIN {X 0,Y 247.194,Z 538.021,A -85,B 0,C 180,E1 -20214.424,E2 -20214.424} C_VEL
LIN {X 0,Y 244.895,Z 541.768,A -85,B 0,C 180,E1 -20215.351,E2 -20215.351} C_VEL
LIN {X 0,Y 244.302,Z 542.937,A -85,B 0,C 180,E1 -20215.696,E2 -20215.696} C_VEL
LIN {X 0,Y 240.466,Z 550.922,A -85,B 0,C 180,E1 -20218.259,E2 -20218.259} C_VEL
LIN {X 0,Y 234.417,Z 561.158,A -85,B 0,C 180,E1 -20221.822,E2 -20221.822} C_VEL
LIN {X 0,Y 230.311,Z 567.866,A -85,B 0,C 180,E1 -20224.709,E2 -20224.709} C_VEL
LIN {X 0,Y 225.836,Z 574.194,A -85,B 0,C 180,E1 -20228.072,E2 -20228.072} C_VEL
LIN {X 0,Y 222.516,Z 579.155,A -85,B 0,C 180,E1 -20231.588,E2 -20231.588} C_VEL
LIN {X 0,Y 220.577,Z 582.823,A -85,B 0,C 180,E1 -20235.232,E2 -20235.232} C_VEL
LIN {X 0,Y 219.882,Z 584.754,A -85,B 0,C 180,E1 -20237.774,E2 -20237.774} C_VEL
LIN {X 0,Y 219.564,Z 588.447,A -85,B 0,C 180,E1 -20240.79,E2 -20240.79} C_VEL
LIN {X 0,Y 219.714,Z 590.176,A -85,B 0,C 180,E1 -20242.649,E2 -20242.649} C_VEL
LIN {X 0,Y 219.973,Z 591.455,A -85,B 0,C 180,E1 -20244.499,E2 -20244.499} C_VEL
LIN {X 0,Y 220.287,Z 592.299,A -85,B 0,C 180,E1 -20246.341,E2 -20246.341} C_VEL
LIN {X 0,Y 221.279,Z 592.798,A -85,B 0,C 180,E1 -20250,E2 -20250} C_VEL
LIN {X 0,Y 220.693,Z 592.245,A -85,B 0,C 180,E1 -20251.825,E2 -20251.825} C_VEL
LIN {X 0,Y 220.351,Z 591.271,A -85,B 0,C 180,E1 -20253.657,E2 -20253.657} C_VEL
LIN {X 0,Y 220.058,Z 589.878,A -85,B 0,C 180,E1 -20255.498,E2 -20255.498} C_VEL
LIN {X 0,Y 219.721,Z 586.939,A -85,B 0,C 180,E1 -20258.274,E2 -20258.274} C_VEL
LIN {X 0,Y 219.749,Z 582.947,A -85,B 0,C 180,E1 -20261.063,E2 -20261.063} C_VEL
LIN {X 0,Y 220.315,Z 577.833,A -85,B 0,C 180,E1 -20263.842,E2 -20263.842} C_VEL
LIN {X 0,Y 221.286,Z 571.423,A -85,B 0,C 180,E1 -20266.609,E2 -20266.609} C_VEL
LIN {X 0,Y 223.15,Z 563.566,A -85,B 0,C 180,E1 -20269.309,E2 -20269.309} C_VEL
LIN {X 0,Y 224.779,Z 555.486,A -85,B 0,C 180,E1 -20271.554,E2 -20271.554} C_VEL
LIN {X 0,Y 225.828,Z 545.489,A -85,B 0,C 180,E1 -20273.864,E2 -20273.864} C_VEL
LIN {X 0,Y 226.62,Z 534.654,A -85,B 0,C 180,E1 -20275.927,E2 -20275.927} C_VEL
LIN {X 0,Y 226.964,Z 523.557,A -85,B 0,C 180,E1 -20277.676,E2 -20277.676} C_VEL
LIN {X 0,Y 226.561,Z 510.814,A -85,B 0,C 180,E1 -20279.336,E2 -20279.336} C_VEL
LIN {X 0,Y 225.297,Z 497.804,A -85,B 0,C 180,E1 -20280.736,E2 -20280.736} C_VEL
LIN {X 0,Y 223.1,Z 484.079,A -85,B 0,C 180,E1 -20281.943,E2 -20281.943} C_VEL
LIN {X 0,Y 222.415,Z 480.111,A -85,B 0,C 180,E1 -20282.246,E2 -20282.246} C_VEL
LIN {X 0,Y 224.084,Z 472.536,A -85,B 0,C 180,E1 -20286.577,E2 -20286.577} C_VEL
LIN {X 0,Y 225.005,Z 468.835,A -85,B 0,C 180,E1 -20288.66,E2 -20288.66} C_VEL
LIN {X 0,Y 225.192,Z 466.964,A -85,B 0,C 180,E1 -20289.775,E2 -20289.775} C_VEL
LIN {X 0,Y 224.492,Z 462.431,A -85,B 0,C 180,E1 -20292.614,E2 -20292.614} C_VEL
LIN {X 0,Y 223.083,Z 455.233,A -85,B 0,C 180,E1 -20297.439,E2 -20297.439} C_VEL
LIN {X 0,Y 221.948,Z 449.295,A -85,B 0,C 180,E1 -20301.717,E2 -20301.717} C_VEL
LIN {X 0,Y 220.852,Z 443.977,A -85,B 0,C 180,E1 -20305.987,E2 -20305.987} C_VEL
LIN {X 0,Y 220.834,Z 443.979,A -85,B 0,C 180,E1 -20309.39,E2 -20309.39} C_VEL
LIN {X 0,Y 220.894,Z 443.968,A -85,B 0,C 180,E1 -20313.55,E2 -20313.55} C_VEL
LIN {X 0,Y 220.924,Z 443.967,A -85,B 0,C 180,E1 -20317.559,E2 -20317.559} C_VEL
LIN {X 0,Y 220.986,Z 443.961,A -85,B 0,C 180,E1 -20322.57,E2 -20322.57} C_VEL
LIN {X 0,Y 221.013,Z 443.955,A -85,B 0,C 180,E1 -20327.139,E2 -20327.139} C_VEL
LIN {X 0,Y 221.202,Z 443.932,A -85,B 0,C 180,E1 -20330.86,E2 -20330.86} C_VEL
LIN {X 0,Y 221.14,Z 443.938,A -85,B 0,C 180,E1 -20334.529,E2 -20334.529} C_VEL
LIN {X 0,Y 221.514,Z 443.892,A -85,B 0,C 180,E1 -20338.182,E2 -20338.182} C_VEL
LIN {X 0,Y 221.514,Z 443.891,A -85,B 0,C 180,E1 -20341.818,E2 -20341.818} C_VEL
LIN {X 0,Y 221.312,Z 443.91,A -85,B 0,C 180,E1 -20347.298,E2 -20347.298} C_VEL
LIN {X 0,Y 221.112,Z 443.939,A -85,B 0,C 180,E1 -20350.994,E2 -20350.994} C_VEL
LIN {X 0,Y 221.018,Z 443.951,A -85,B 0,C 180,E1 -20356.63,E2 -20356.63} C_VEL
LIN {X 0,Y 220.894,Z 443.947,A -85,B 0,C 180,E1 -20360.486,E2 -20360.486} C_VEL
LIN {X 0,Y 220.869,Z 443.954,A -85,B 0,C 180,E1 -20364.435,E2 -20364.435} C_VEL
LIN {X 0,Y 220.837,Z 443.975,A -85,B 0,C 180,E1 -20368.514,E2 -20368.514} C_VEL
LIN {X 0,Y 220.825,Z 443.952,A -85,B 0,C 180,E1 -20372.755,E2 -20372.755} C_VEL
LIN {X 0,Y 220.839,Z 443.975,A -85,B 0,C 180,E1 -20377.288,E2 -20377.288} C_VEL
LIN {X 0,Y 220.776,Z 443.984,A -85,B 0,C 180,E1 -20381.952,E2 -20381.952} C_VEL
LIN {X 0,Y 220.775,Z 443.979,A -85,B 0,C 180,E1 -20385.547,E2 -20385.547} C_VEL
LIN {X 0,Y 220.811,Z 443.974,A -85,B 0,C 180,E1 -20390.464,E2 -20390.464} C_VEL
LIN {X 0,Y 220.833,Z 443.971,A -85,B 0,C 180,E1 -20392.795,E2 -20392.795} C_VEL
LIN {X 0,Y 220.827,Z 443.973,A -85,B 0,C 180,E1 -20397.246,E2 -20397.246} C_VEL
LIN {X 0,Y 220.84,Z 443.964,A -85,B 0,C 180,E1 -20401.487,E2 -20401.487} C_VEL
LIN {X 0,Y 220.851,Z 444.005,A -85,B 0,C 180,E1 -20401.855,E2 -20401.855} C_VEL
LIN {X 0,Y 221.12,Z 445.23,A -85,B 0,C 180,E1 -20402.008,E2 -20402.008} C_VEL
LIN {X 0,Y 225.916,Z 455.718,A -85,B 0,C 180,E1 -20403.928,E2 -20403.928} C_VEL
LIN {X 0,Y 229.647,Z 466.07,A -85,B 0,C 180,E1 -20405.952,E2 -20405.952} C_VEL
LIN {X 0,Y 232.398,Z 475.684,A -85,B 0,C 180,E1 -20408.02,E2 -20408.02} C_VEL
LIN {X 0,Y 233.342,Z 480.012,A -85,B 0,C 180,E1 -20409.018,E2 -20409.018} C_VEL
LIN {X 0,Y 231.431,Z 489.434,A -85,B 0,C 180,E1 -20410.947,E2 -20410.947} C_VEL
LIN {X 0,Y 229.354,Z 497.94,A -85,B 0,C 180,E1 -20413.076,E2 -20413.076} C_VEL
LIN {X 0,Y 227.228,Z 506.181,A -85,B 0,C 180,E1 -20415.675,E2 -20415.675} C_VEL
LIN {X 0,Y 225.511,Z 512.788,A -85,B 0,C 180,E1 -20418.313,E2 -20418.313} C_VEL
LIN {X 0,Y 224.139,Z 518.063,A -85,B 0,C 180,E1 -20420.98,E2 -20420.98} C_VEL
LIN {X 0,Y 222.935,Z 522.213,A -85,B 0,C 180,E1 -20423.666,E2 -20423.666} C_VEL
LIN {X 0,Y 222.013,Z 525.337,A -85,B 0,C 180,E1 -20426.37,E2 -20426.37} C_VEL
LIN {X 0,Y 221.519,Z 528.026,A -85,B 0,C 180,E1 -20430,E2 -20430} C_VEL
LIN {X 0,Y 221.513,Z 528.739,A -85,B 0,C 180,E1 -20431.819,E2 -20431.819} C_VEL
LIN {X 0,Y 221.447,Z 529.117,A -85,B 0,C 180,E1 -20435.464,E2 -20435.464} C_VEL
LIN {X 0,Y 221.851,Z 528.711,A -85,B 0,C 180,E1 -20437.28,E2 -20437.28} C_VEL
LIN {X 0,Y 223.267,Z 526.635,A -85,B 0,C 180,E1 -20440.887,E2 -20440.887} C_VEL
LIN {X 0,Y 224.713,Z 523.39,A -85,B 0,C 180,E1 -20444.176,E2 -20444.176} C_VEL
LIN {X 0,Y 226.399,Z 519.107,A -85,B 0,C 180,E1 -20447.152,E2 -20447.152} C_VEL
LIN {X 0,Y 228.224,Z 514.047,A -85,B 0,C 180,E1 -20449.8,E2 -20449.8} C_VEL
LIN {X 0,Y 230.35,Z 507.663,A -85,B 0,C 180,E1 -20452.419,E2 -20452.419} C_VEL
LIN {X 0,Y 232.984,Z 499.671,A -85,B 0,C 180,E1 -20454.981,E2 -20454.981} C_VEL
LIN {X 0,Y 235.36,Z 491.476,A -85,B 0,C 180,E1 -20457.09,E2 -20457.09} C_VEL
LIN {X 0,Y 236.289,Z 487.696,A -85,B 0,C 180,E1 -20457.935,E2 -20457.935} C_VEL
LIN {X 0,Y 236.416,Z 485.721,A -85,B 0,C 180,E1 -20458.401,E2 -20458.401} C_VEL
LIN {X 0,Y 234.469,Z 477.111,A -85,B 0,C 180,E1 -20460.635,E2 -20460.635} C_VEL
LIN {X 0,Y 231.348,Z 467.358,A -85,B 0,C 180,E1 -20462.982,E2 -20462.982} C_VEL
LIN {X 0,Y 227.437,Z 457.78,A -85,B 0,C 180,E1 -20465.155,E2 -20465.155} C_VEL
LIN {X 0,Y 224.66,Z 451.717,A -85,B 0,C 180,E1 -20466.469,E2 -20466.469} C_VEL
LIN {X 0,Y 221.159,Z 445.369,A -85,B 0,C 180,E1 -20467.856,E2 -20467.856} C_VEL
LIN {X 0,Y 220.829,Z 443.978,A -85,B 0,C 180,E1 -20468.115,E2 -20468.115} C_VEL
LIN {X 0,Y 220.772,Z 443.984,A -85,B 0,C 180,E1 -20472.93,E2 -20472.93} C_VEL
LIN {X 0,Y 220.772,Z 443.979,A -85,B 0,C 180,E1 -20477.07,E2 -20477.07} C_VEL
LIN {X 0,Y 220.813,Z 443.974,A -85,B 0,C 180,E1 -20480.464,E2 -20480.464} C_VEL
LIN {X 0,Y 220.835,Z 443.975,A -85,B 0,C 180,E1 -20482.794,E2 -20482.794} C_VEL
LIN {X 0,Y 220.828,Z 443.975,A -85,B 0,C 180,E1 -20487.245,E2 -20487.245} C_VEL
LIN {X 0,Y 220.84,Z 443.972,A -85,B 0,C 180,E1 -20491.487,E2 -20491.487} C_VEL
LIN {X 0,Y 220.866,Z 443.969,A -85,B 0,C 180,E1 -20495.564,E2 -20495.564} C_VEL
LIN {X 0,Y 221.035,Z 444.035,A -85,B 0,C 180,E1 -20499.909,E2 -20499.909} C_VEL
LIN {X 0,Y 224.006,Z 457.616,A -85,B 0,C 180,E1 -20501.715,E2 -20501.715} C_VEL
LIN {X 0,Y 224.906,Z 462.754,A -85,B 0,C 180,E1 -20502.496,E2 -20502.496} C_VEL
LIN {X 0,Y 223.948,Z 474.74,A -85,B 0,C 180,E1 -20504.529,E2 -20504.529} C_VEL
LIN {X 0,Y 222.875,Z 485.732,A -85,B 0,C 180,E1 -20506.784,E2 -20506.784} C_VEL
LIN {X 0,Y 221.917,Z 496.035,A -85,B 0,C 180,E1 -20509.355,E2 -20509.355} C_VEL
LIN {X 0,Y 221.331,Z 504.144,A -85,B 0,C 180,E1 -20511.785,E2 -20511.785} C_VEL
LIN {X 0,Y 220.697,Z 511.761,A -85,B 0,C 180,E1 -20514.518,E2 -20514.518} C_VEL
LIN {X 0,Y 220.741,Z 518.104,A -85,B 0,C 180,E1 -20517.262,E2 -20517.262} C_VEL
LIN {X 0,Y 221.178,Z 524.8,A -85,B 0,C 180,E1 -20520.91,E2 -20520.91} C_VEL
LIN {X 0,Y 221.715,Z 528.649,A -85,B 0,C 180,E1 -20523.635,E2 -20523.635} C_VEL
LIN {X 0,Y 222.335,Z 530.744,A -85,B 0,C 180,E1 -20525.441,E2 -20525.441} C_VEL
LIN {X 0,Y 224.122,Z 533.721,A -85,B 0,C 180,E1 -20529.02,E2 -20529.02} C_VEL
LIN {X 0,Y 226.871,Z 535.221,A -85,B 0,C 180,E1 -20532.524,E2 -20532.524} C_VEL
LIN {X 0,Y 230.209,Z 535.235,A -85,B 0,C 180,E1 -20535.947,E2 -20535.947} C_VEL
LIN {X 0,Y 234.379,Z 533.855,A -85,B 0,C 180,E1 -20539.259,E2 -20539.259} C_VEL
LIN {X 0,Y 239.275,Z 530.981,A -85,B 0,C 180,E1 -20542.447,E2 -20542.447} C_VEL
LIN {X 0,Y 244.901,Z 526.629,A -85,B 0,C 180,E1 -20545.497,E2 -20545.497} C_VEL
LIN {X 0,Y 251.187,Z 520.617,A -85,B 0,C 180,E1 -20548.401,E2 -20548.401} C_VEL
LIN {X 0,Y 257.209,Z 513.883,A -85,B 0,C 180,E1 -20550.819,E2 -20550.819} C_VEL
LIN {X 0,Y 258.109,Z 512.787,A -85,B 0,C 180,E1 -20551.154,E2 -20551.154} C_VEL
LIN {X 0,Y 258.732,Z 511.655,A -85,B 0,C 180,E1 -20551.77,E2 -20551.77} C_VEL
LIN {X 0,Y 259.665,Z 509.116,A -85,B 0,C 180,E1 -20553.525,E2 -20553.525} C_VEL
LIN {X 0,Y 260.337,Z 506.528,A -85,B 0,C 180,E1 -20555.915,E2 -20555.915} C_VEL
LIN {X 0,Y 260.095,Z 505.586,A -85,B 0,C 180,E1 -20558.424,E2 -20558.424} C_VEL
LIN {X 0,Y 259.434,Z 506.196,A -85,B 0,C 180,E1 -20560.666,E2 -20560.666} C_VEL
LIN {X 0,Y 258.665,Z 507.947,A -85,B 0,C 180,E1 -20562.811,E2 -20562.811} C_VEL
LIN {X 0,Y 257.441,Z 511.465,A -85,B 0,C 180,E1 -20565.217,E2 -20565.217} C_VEL
LIN {X 0,Y 256.424,Z 513.78,A -85,B 0,C 180,E1 -20566.199,E2 -20566.199} C_VEL
LIN {X 0,Y 253.816,Z 519.89,A -85,B 0,C 180,E1 -20568.384,E2 -20568.384} C_VEL
LIN {X 0,Y 249.038,Z 531.735,A -85,B 0,C 180,E1 -20572.202,E2 -20572.202} C_VEL
LIN {X 0,Y 245.224,Z 540.822,A -85,B 0,C 180,E1 -20575.027,E2 -20575.027} C_VEL
LIN {X 0,Y 244.302,Z 542.937,A -85,B 0,C 180,E1 -20575.696,E2 -20575.696} C_VEL
LIN {X 0,Y 242.084,Z 546.552,A -85,B 0,C 180,E1 -20576.679,E2 -20576.679} C_VEL
LIN {X 0,Y 236.743,Z 552.555,A -85,B 0,C 180,E1 -20578.093,E2 -20578.093} C_VEL
LIN {X 0,Y 231.172,Z 558.093,A -85,B 0,C 180,E1 -20579.592,E2 -20579.592} C_VEL
LIN {X 0,Y 228.655,Z 561.091,A -85,B 0,C 180,E1 -20580.698,E2 -20580.698} C_VEL
LIN {X 0,Y 223.904,Z 568.056,A -85,B 0,C 180,E1 -20583.931,E2 -20583.931} C_VEL
LIN {X 0,Y 219.234,Z 574.002,A -85,B 0,C 180,E1 -20587.375,E2 -20587.375} C_VEL
LIN {X 0,Y 215.738,Z 578.567,A -85,B 0,C 180,E1 -20590.988,E2 -20590.988} C_VEL
LIN {X 0,Y 213.681,Z 581.889,A -85,B 0,C 180,E1 -20594.744,E2 -20594.744} C_VEL
LIN {X 0,Y 212.972,Z 583.456,A -85,B 0,C 180,E1 -20597.129,E2 -20597.129} C_VEL
LIN {X 0,Y 212.51,Z 587.46,A -85,B 0,C 180,E1 -20600.482,E2 -20600.482} C_VEL
LIN {X 0,Y 212.626,Z 589.309,A -85,B 0,C 180,E1 -20602.568,E2 -20602.568} C_VEL
LIN {X 0,Y 212.875,Z 590.447,A -85,B 0,C 180,E1 -20604.315,E2 -20604.315} C_VEL
LIN {X 0,Y 213.223,Z 591.29,A -85,B 0,C 180,E1 -20606.22,E2 -20606.22} C_VEL
LIN {X 0,Y 214.236,Z 591.78,A -85,B 0,C 180,E1 -20610,E2 -20610} C_VEL
LIN {X 0,Y 213.627,Z 591.207,A -85,B 0,C 180,E1 -20611.885,E2 -20611.885} C_VEL
LIN {X 0,Y 213.286,Z 590.224,A -85,B 0,C 180,E1 -20613.778,E2 -20613.778} C_VEL
LIN {X 0,Y 212.961,Z 588.816,A -85,B 0,C 180,E1 -20615.681,E2 -20615.681} C_VEL
LIN {X 0,Y 212.66,Z 585.859,A -85,B 0,C 180,E1 -20618.551,E2 -20618.551} C_VEL
LIN {X 0,Y 212.717,Z 581.845,A -85,B 0,C 180,E1 -20621.433,E2 -20621.433} C_VEL
LIN {X 0,Y 213.329,Z 576.706,A -85,B 0,C 180,E1 -20624.305,E2 -20624.305} C_VEL
LIN {X 0,Y 214.427,Z 570.282,A -85,B 0,C 180,E1 -20627.156,E2 -20627.156} C_VEL
LIN {X 0,Y 216.39,Z 562.388,A -85,B 0,C 180,E1 -20629.938,E2 -20629.938} C_VEL
LIN {X 0,Y 217.759,Z 556.013,A -85,B 0,C 180,E1 -20631.786,E2 -20631.786} C_VEL
LIN {X 0,Y 218.883,Z 546.429,A -85,B 0,C 180,E1 -20634.166,E2 -20634.166} C_VEL
LIN {X 0,Y 219.743,Z 536.666,A -85,B 0,C 180,E1 -20636.167,E2 -20636.167} C_VEL
LIN {X 0,Y 220.241,Z 525.463,A -85,B 0,C 180,E1 -20638.078,E2 -20638.078} C_VEL
LIN {X 0,Y 220.062,Z 512.613,A -85,B 0,C 180,E1 -20639.897,E2 -20639.897} C_VEL
LIN {X 0,Y 219.014,Z 499.798,A -85,B 0,C 180,E1 -20641.405,E2 -20641.405} C_VEL
LIN {X 0,Y 216.973,Z 485.97,A -85,B 0,C 180,E1 -20642.731,E2 -20642.731} C_VEL
LIN {X 0,Y 215.694,Z 479.097,A -85,B 0,C 180,E1 -20643.294,E2 -20643.294} C_VEL
LIN {X 0,Y 217.552,Z 471.347,A -85,B 0,C 180,E1 -20647.864,E2 -20647.864} C_VEL
LIN {X 0,Y 218.13,Z 467.602,A -85,B 0,C 180,E1 -20650.119,E2 -20650.119} C_VEL
LIN {X 0,Y 217.217,Z 462.2,A -85,B 0,C 180,E1 -20653.651,E2 -20653.651} C_VEL
LIN {X 0,Y 215.893,Z 455.356,A -85,B 0,C 180,E1 -20658.479,E2 -20658.479} C_VEL
LIN {X 0,Y 214.826,Z 449.66,A -85,B 0,C 180,E1 -20662.763,E2 -20662.763} C_VEL
LIN {X 0,Y 213.821,Z 444.856,A -85,B 0,C 180,E1 -20666.736,E2 -20666.736} C_VEL
LIN {X 0,Y 213.76,Z 444.858,A -85,B 0,C 180,E1 -20670.451,E2 -20670.451} C_VEL
LIN {X 0,Y 213.805,Z 444.853,A -85,B 0,C 180,E1 -20674.702,E2 -20674.702} C_VEL
LIN {X 0,Y 213.841,Z 444.851,A -85,B 0,C 180,E1 -20678.807,E2 -20678.807} C_VEL
LIN {X 0,Y 213.945,Z 444.838,A -85,B 0,C 180,E1 -20682.804,E2 -20682.804} C_VEL
LIN {X 0,Y 213.954,Z 444.835,A -85,B 0,C 180,E1 -20686.707,E2 -20686.707} C_VEL
LIN {X 0,Y 214.14,Z 444.813,A -85,B 0,C 180,E1 -20690.555,E2 -20690.555} C_VEL
LIN {X 0,Y 214.101,Z 444.816,A -85,B 0,C 180,E1 -20694.349,E2 -20694.349} C_VEL
LIN {X 0,Y 214.448,Z 444.772,A -85,B 0,C 180,E1 -20698.122,E2 -20698.122} C_VEL
LIN {X 0,Y 214.556,Z 444.76,A -85,B 0,C 180,E1 -20700,E2 -20700} C_VEL
LIN {X 0,Y 214.447,Z 444.772,A -85,B 0,C 180,E1 -20701.878,E2 -20701.878} C_VEL
LIN {X 0,Y 214.249,Z 444.79,A -85,B 0,C 180,E1 -20707.54,E2 -20707.54} C_VEL
LIN {X 0,Y 214.043,Z 444.82,A -85,B 0,C 180,E1 -20711.362,E2 -20711.362} C_VEL
LIN {X 0,Y 213.935,Z 444.833,A -85,B 0,C 180,E1 -20715.237,E2 -20715.237} C_VEL
LIN {X 0,Y 213.841,Z 444.836,A -85,B 0,C 180,E1 -20719.188,E2 -20719.188} C_VEL
LIN {X 0,Y 213.848,Z 444.816,A -85,B 0,C 180,E1 -20723.227,E2 -20723.227} C_VEL
LIN {X 0,Y 213.83,Z 444.848,A -85,B 0,C 180,E1 -20727.45,E2 -20727.45} C_VEL
LIN {X 0,Y 213.78,Z 444.835,A -85,B 0,C 180,E1 -20731.736,E2 -20731.736} C_VEL
LIN {X 0,Y 213.754,Z 444.854,A -85,B 0,C 180,E1 -20736.287,E2 -20736.287} C_VEL
LIN {X 0,Y 213.717,Z 444.858,A -85,B 0,C 180,E1 -20741.125,E2 -20741.125} C_VEL
LIN {X 0,Y 213.709,Z 444.859,A -85,B 0,C 180,E1 -20743.679,E2 -20743.679} C_VEL
LIN {X 0,Y 213.709,Z 444.86,A -85,B 0,C 180,E1 -20746.344,E2 -20746.344} C_VEL
LIN {X 0,Y 213.738,Z 444.853,A -85,B 0,C 180,E1 -20751.337,E2 -20751.337} C_VEL
LIN {X 0,Y 213.772,Z 444.854,A -85,B 0,C 180,E1 -20756.021,E2 -20756.021} C_VEL
LIN {X 0,Y 213.797,Z 444.857,A -85,B 0,C 180,E1 -20760.737,E2 -20760.737} C_VEL
LIN {X 0,Y 214.462,Z 447.113,A -85,B 0,C 180,E1 -20761.072,E2 -20761.072} C_VEL
LIN {X 0,Y 219.054,Z 456.851,A -85,B 0,C 180,E1 -20762.983,E2 -20762.983} C_VEL
LIN {X 0,Y 222.69,Z 466.723,A -85,B 0,C 180,E1 -20765.011,E2 -20765.011} C_VEL
LIN {X 0,Y 225.715,Z 477.193,A -85,B 0,C 180,E1 -20767.367,E2 -20767.367} C_VEL
LIN {X 0,Y 226.694,Z 481.657,A -85,B 0,C 180,E1 -20768.447,E2 -20768.447} C_VEL
LIN {X 0,Y 224.828,Z 490.664,A -85,B 0,C 180,E1 -20770.365,E2 -20770.365} C_VEL
LIN {X 0,Y 222.664,Z 499.132,A -85,B 0,C 180,E1 -20772.552,E2 -20772.552} C_VEL
LIN {X 0,Y 220.445,Z 507.331,A -85,B 0,C 180,E1 -20775.224,E2 -20775.224} C_VEL
LIN {X 0,Y 218.648,Z 513.912,A -85,B 0,C 180,E1 -20777.941,E2 -20777.941} C_VEL
LIN {X 0,Y 217.212,Z 519.165,A -85,B 0,C 180,E1 -20780.69,E2 -20780.69} C_VEL
LIN {X 0,Y 215.98,Z 523.292,A -85,B 0,C 180,E1 -20783.461,E2 -20783.461} C_VEL
LIN {X 0,Y 215.004,Z 526.4,A -85,B 0,C 180,E1 -20786.252,E2 -20786.252} C_VEL
LIN {X 0,Y 214.653,Z 527.936,A -85,B 0,C 180,E1 -20788.124,E2 -20788.124} C_VEL
LIN {X 0,Y 214.492,Z 529.063,A -85,B 0,C 180,E1 -20790,E2 -20790} C_VEL
LIN {X 0,Y 214.488,Z 529.765,A -85,B 0,C 180,E1 -20791.878,E2 -20791.878} C_VEL
LIN {X 0,Y 214.446,Z 530.125,A -85,B 0,C 180,E1 -20795.643,E2 -20795.643} C_VEL
LIN {X 0,Y 214.876,Z 529.704,A -85,B 0,C 180,E1 -20797.518,E2 -20797.518} C_VEL
LIN {X 0,Y 216.367,Z 527.606,A -85,B 0,C 180,E1 -20801.239,E2 -20801.239} C_VEL
LIN {X 0,Y 217.904,Z 524.342,A -85,B 0,C 180,E1 -20804.627,E2 -20804.627} C_VEL
LIN {X 0,Y 219.677,Z 520.029,A -85,B 0,C 180,E1 -20807.694,E2 -20807.694} C_VEL
LIN {X 0,Y 221.613,Z 514.945,A -85,B 0,C 180,E1 -20810.417,E2 -20810.417} C_VEL
LIN {X 0,Y 223.856,Z 508.537,A -85,B 0,C 180,E1 -20813.107,E2 -20813.107} C_VEL
LIN {X 0,Y 226.615,Z 500.516,A -85,B 0,C 180,E1 -20815.734,E2 -20815.734} C_VEL
LIN {X 0,Y 229.105,Z 492.288,A -85,B 0,C 180,E1 -20817.893,E2 -20817.893} C_VEL
LIN {X 0,Y 229.959,Z 488.504,A -85,B 0,C 180,E1 -20818.774,E2 -20818.774} C_VEL
LIN {X 0,Y 228.684,Z 481.788,A -85,B 0,C 180,E1 -20820.626,E2 -20820.626} C_VEL
LIN {X 0,Y 226.141,Z 472.84,A -85,B 0,C 180,E1 -20822.953,E2 -20822.953} C_VEL
LIN {X 0,Y 222.585,Z 463.364,A -85,B 0,C 180,E1 -20825.283,E2 -20825.283} C_VEL
LIN {X 0,Y 218.51,Z 454.524,A -85,B 0,C 180,E1 -20827.375,E2 -20827.375} C_VEL
LIN {X 0,Y 215.844,Z 449.074,A -85,B 0,C 180,E1 -20828.605,E2 -20828.605} C_VEL
LIN {X 0,Y 214.068,Z 446.207,A -85,B 0,C 180,E1 -20829.303,E2 -20829.303} C_VEL
LIN {X 0,Y 213.781,Z 444.856,A -85,B 0,C 180,E1 -20829.534,E2 -20829.534} C_VEL
LIN {X 0,Y 213.711,Z 444.861,A -85,B 0,C 180,E1 -20833.678,E2 -20833.678} C_VEL
LIN {X 0,Y 213.711,Z 444.862,A -85,B 0,C 180,E1 -20836.344,E2 -20836.344} C_VEL
LIN {X 0,Y 213.74,Z 444.856,A -85,B 0,C 180,E1 -20841.336,E2 -20841.336} C_VEL
LIN {X 0,Y 213.774,Z 444.857,A -85,B 0,C 180,E1 -20846.02,E2 -20846.02} C_VEL
LIN {X 0,Y 213.784,Z 444.853,A -85,B 0,C 180,E1 -20850.454,E2 -20850.454} C_VEL
LIN {X 0,Y 213.802,Z 444.85,A -85,B 0,C 180,E1 -20854.701,E2 -20854.701} C_VEL
LIN {X 0,Y 213.986,Z 444.956,A -85,B 0,C 180,E1 -20859.796,E2 -20859.796} C_VEL
LIN {X 0,Y 216.835,Z 457.979,A -85,B 0,C 180,E1 -20861.578,E2 -20861.578} C_VEL
LIN {X 0,Y 217.807,Z 463.204,A -85,B 0,C 180,E1 -20862.392,E2 -20862.392} C_VEL
LIN {X 0,Y 216.813,Z 475.324,A -85,B 0,C 180,E1 -20864.489,E2 -20864.489} C_VEL
LIN {X 0,Y 215.762,Z 486.365,A -85,B 0,C 180,E1 -20866.82,E2 -20866.82} C_VEL
LIN {X 0,Y 214.824,Z 495.982,A -85,B 0,C 180,E1 -20869.276,E2 -20869.276} C_VEL
LIN {X 0,Y 214.181,Z 504.821,A -85,B 0,C 180,E1 -20871.983,E2 -20871.983} C_VEL
LIN {X 0,Y 213.583,Z 513.713,A -85,B 0,C 180,E1 -20875.281,E2 -20875.281} C_VEL
LIN {X 0,Y 213.632,Z 519.92,A -85,B 0,C 180,E1 -20878.114,E2 -20878.114} C_VEL
LIN {X 0,Y 214.097,Z 524.992,A -85,B 0,C 180,E1 -20880.94,E2 -20880.94} C_VEL
LIN {X 0,Y 214.974,Z 530.278,A -85,B 0,C 180,E1 -20884.688,E2 -20884.688} C_VEL
LIN {X 0,Y 216.139,Z 533.181,A -85,B 0,C 180,E1 -20887.473,E2 -20887.473} C_VEL
LIN {X 0,Y 217.198,Z 534.663,A -85,B 0,C 180,E1 -20889.31,E2 -20889.31} C_VEL
LIN {X 0,Y 220.076,Z 536.439,A -85,B 0,C 180,E1 -20892.917,E2 -20892.917} C_VEL
LIN {X 0,Y 223.578,Z 536.841,A -85,B 0,C 180,E1 -20896.434,E2 -20896.434} C_VEL
LIN {X 0,Y 227.938,Z 535.768,A -85,B 0,C 180,E1 -20899.826,E2 -20899.826} C_VEL
LIN {X 0,Y 233.091,Z 533.322,A -85,B 0,C 180,E1 -20903.077,E2 -20903.077} C_VEL
LIN {X 0,Y 238.96,Z 529.376,A -85,B 0,C 180,E1 -20906.178,E2 -20906.178} C_VEL
LIN {X 0,Y 245.531,Z 523.868,A -85,B 0,C 180,E1 -20909.117,E2 -20909.117} C_VEL
LIN {X 0,Y 251.81,Z 517.603,A -85,B 0,C 180,E1 -20911.555,E2 -20911.555} C_VEL
LIN {X 0,Y 252.74,Z 516.601,A -85,B 0,C 180,E1 -20911.893,E2 -20911.893} C_VEL
LIN {X 0,Y 253.559,Z 515.475,A -85,B 0,C 180,E1 -20912.496,E2 -20912.496} C_VEL
LIN {X 0,Y 254.572,Z 513.456,A -85,B 0,C 180,E1 -20914.083,E2 -20914.083} C_VEL
LIN {X 0,Y 255.129,Z 512.219,A -85,B 0,C 180,E1 -20915.344,E2 -20915.344} C_VEL
LIN {X 0,Y 255.35,Z 511.141,A -85,B 0,C 180,E1 -20917.265,E2 -20917.265} C_VEL
LIN {X 0,Y 255.021,Z 511.162,A -85,B 0,C 180,E1 -20919.498,E2 -20919.498} C_VEL
LIN {X 0,Y 254.258,Z 512.502,A -85,B 0,C 180,E1 -20921.727,E2 -20921.727} C_VEL
LIN {X 0,Y 253.884,Z 513.392,A -85,B 0,C 180,E1 -20922.696,E2 -20922.696} C_VEL
LIN {X 0,Y 253.184,Z 515.077,A -85,B 0,C 180,E1 -20923.944,E2 -20923.944} C_VEL
LIN {X 0,Y 252.407,Z 516.927,A -85,B 0,C 180,E1 -20925.017,E2 -20925.017} C_VEL
LIN {X 0,Y 249.205,Z 523.173,A -85,B 0,C 180,E1 -20927.402,E2 -20927.402} C_VEL
LIN {X 0,Y 243.847,Z 534.284,A -85,B 0,C 180,E1 -20931.25,E2 -20931.25} C_VEL
LIN {X 0,Y 239.067,Z 543.987,A -85,B 0,C 180,E1 -20934.506,E2 -20934.506} C_VEL
LIN {X 0,Y 234.573,Z 552.232,A -85,B 0,C 180,E1 -20937.364,E2 -20937.364} C_VEL
LIN {X 0,Y 228.655,Z 561.091,A -85,B 0,C 180,E1 -20940.698,E2 -20940.698} C_VEL
LIN {X 0,Y 226.125,Z 563.968,A -85,B 0,C 180,E1 -20941.845,E2 -20941.845} C_VEL
LIN {X 0,Y 220.386,Z 568.348,A -85,B 0,C 180,E1 -20943.61,E2 -20943.61} C_VEL
LIN {X 0,Y 214.741,Z 572.053,A -85,B 0,C 180,E1 -20945.521,E2 -20945.521} C_VEL
LIN {X 0,Y 212.413,Z 573.997,A -85,B 0,C 180,E1 -20946.876,E2 -20946.876} C_VEL
LIN {X 0,Y 208.996,Z 577.924,A -85,B 0,C 180,E1 -20950.349,E2 -20950.349} C_VEL
LIN {X 0,Y 206.805,Z 580.933,A -85,B 0,C 180,E1 -20954.224,E2 -20954.224} C_VEL
LIN {X 0,Y 206.095,Z 582.157,A -85,B 0,C 180,E1 -20956.441,E2 -20956.441} C_VEL
LIN {X 0,Y 205.456,Z 586.473,A -85,B 0,C 180,E1 -20960.152,E2 -20960.152} C_VEL
LIN {X 0,Y 205.581,Z 588.422,A -85,B 0,C 180,E1 -20962.478,E2 -20962.478} C_VEL
LIN {X 0,Y 206.157,Z 590.282,A -85,B 0,C 180,E1 -20966.09,E2 -20966.09} C_VEL
LIN {X 0,Y 207.192,Z 590.762,A -85,B 0,C 180,E1 -20970,E2 -20970} C_VEL
LIN {X 0,Y 206.56,Z 590.169,A -85,B 0,C 180,E1 -20971.949,E2 -20971.949} C_VEL
LIN {X 0,Y 206.219,Z 589.177,A -85,B 0,C 180,E1 -20973.908,E2 -20973.908} C_VEL
LIN {X 0,Y 205.658,Z 586.078,A -85,B 0,C 180,E1 -20977.684,E2 -20977.684} C_VEL
LIN {X 0,Y 205.586,Z 582.228,A -85,B 0,C 180,E1 -20980.837,E2 -20980.837} C_VEL
LIN {X 0,Y 206.08,Z 577.461,A -85,B 0,C 180,E1 -20983.811,E2 -20983.811} C_VEL
LIN {X 0,Y 207.056,Z 571.448,A -85,B 0,C 180,E1 -20986.768,E2 -20986.768} C_VEL
LIN {X 0,Y 208.957,Z 564.034,A -85,B 0,C 180,E1 -20989.653,E2 -20989.653} C_VEL
LIN {X 0,Y 210.742,Z 556.496,A -85,B 0,C 180,E1 -20992.035,E2 -20992.035} C_VEL
LIN {X 0,Y 212.056,Z 546.197,A -85,B 0,C 180,E1 -20994.734,E2 -20994.734} C_VEL
LIN {X 0,Y 213.069,Z 535.318,A -85,B 0,C 180,E1 -20997.053,E2 -20997.053} C_VEL
LIN {X 0,Y 213.595,Z 524.039,A -85,B 0,C 180,E1 -20999.033,E2 -20999.033} C_VEL
LIN {X 0,Y 213.4,Z 511.223,A -85,B 0,C 180,E1 -21000.911,E2 -21000.911} C_VEL
LIN {X 0,Y 212.426,Z 499.132,A -85,B 0,C 180,E1 -21002.395,E2 -21002.395} C_VEL
LIN {X 0,Y 210.418,Z 485.587,A -85,B 0,C 180,E1 -21003.779,E2 -21003.779} C_VEL
LIN {X 0,Y 209.03,Z 477.981,A -85,B 0,C 180,E1 -21004.44,E2 -21004.44} C_VEL
LIN {X 0,Y 210.982,Z 470.138,A -85,B 0,C 180,E1 -21009.264,E2 -21009.264} C_VEL
LIN {X 0,Y 211.007,Z 467.712,A -85,B 0,C 180,E1 -21010.816,E2 -21010.816} C_VEL
LIN {X 0,Y 209.803,Z 461.264,A -85,B 0,C 180,E1 -21015.295,E2 -21015.295} C_VEL
LIN {X 0,Y 208.553,Z 454.683,A -85,B 0,C 180,E1 -21020.188,E2 -21020.188} C_VEL
LIN {X 0,Y 207.533,Z 449.475,A -85,B 0,C 180,E1 -21024.365,E2 -21024.365} C_VEL
LIN {X 0,Y 206.739,Z 445.735,A -85,B 0,C 180,E1 -21027.717,E2 -21027.717} C_VEL
LIN {X 0,Y 206.764,Z 445.728,A -85,B 0,C 180,E1 -21032.098,E2 -21032.098} C_VEL
LIN {X 0,Y 206.793,Z 445.727,A -85,B 0,C 180,E1 -21036.579,E2 -21036.579} C_VEL
LIN {X 0,Y 206.879,Z 445.719,A -85,B 0,C 180,E1 -21042.197,E2 -21042.197} C_VEL
LIN {X 0,Y 206.897,Z 445.717,A -85,B 0,C 180,E1 -21046.245,E2 -21046.245} C_VEL
LIN {X 0,Y 207.099,Z 445.69,A -85,B 0,C 180,E1 -21050.231,E2 -21050.231} C_VEL
LIN {X 0,Y 207.062,Z 445.694,A -85,B 0,C 180,E1 -21054.156,E2 -21054.156} C_VEL
LIN {X 0,Y 207.384,Z 445.652,A -85,B 0,C 180,E1 -21058.058,E2 -21058.058} C_VEL
LIN {X 0,Y 207.52,Z 445.637,A -85,B 0,C 180,E1 -21060,E2 -21060} C_VEL
LIN {X 0,Y 207.088,Z 445.688,A -85,B 0,C 180,E1 -21063.892,E2 -21063.892} C_VEL
